LIN {X 0,Y 397.096,Z 510.019,A -85,B 0,C 180,E1 -11203.649,E2 -11203.649} C_VEL
LIN {X 0,Y 397.1,Z 510.023,A -85,B 0,C 180,E1 -11206.521,E2 -11206.521} C_VEL
LIN {X 0,Y 397.111,Z 510.021,A -85,B 0,C 180,E1 -11210.424,E2 -11210.424} C_VEL
LIN {X 0,Y 397.107,Z 510.02,A -85,B 0,C 180,E1 -11214.266,E2 -11214.266} C_VEL
LIN {X 0,Y 397.113,Z 510.025,A -85,B 0,C 180,E1 -11216.728,E2 -11216.728} C_VEL
LIN {X 0,Y 397.129,Z 510.185,A -85,B 0,C 180,E1 -11218.395,E2 -11218.395} C_VEL
LIN {X 0,Y 399.849,Z 521.047,A -85,B 0,C 180,E1 -11221.067,E2 -11221.067} C_VEL
LIN {X 0,Y 401.622,Z 530.428,A -85,B 0,C 180,E1 -11223.183,E2 -11223.183} C_VEL
LIN {X 0,Y 401.493,Z 534.696,A -85,B 0,C 180,E1 -11224.049,E2 -11224.049} C_VEL
LIN {X 0,Y 399.863,Z 552.668,A -85,B 0,C 180,E1 -11227.526,E2 -11227.526} C_VEL
LIN {X 0,Y 399.207,Z 561.982,A -85,B 0,C 180,E1 -11229.268,E2 -11229.268} C_VEL
LIN {X 0,Y 402.568,Z 583.232,A -85,B 0,C 180,E1 -11230.004,E2 -11230.004} C_VEL
LIN {X 0,Y 404.122,Z 598.929,A -85,B 0,C 180,E1 -11230.474,E2 -11230.474} C_VEL
LIN {X 0,Y 402.335,Z 674.306,A -85,B 0,C 180,E1 -11232.135,E2 -11232.135} C_VEL
LIN {X 0,Y 401.685,Z 687.799,A -85,B 0,C 180,E1 -11232.631,E2 -11232.631} C_VEL
LIN {X 0,Y 400.492,Z 707.778,A -85,B 0,C 180,E1 -11233.694,E2 -11233.694} C_VEL
LIN {X 0,Y 399.642,Z 720.158,A -85,B 0,C 180,E1 -11234.575,E2 -11234.575} C_VEL
LIN {X 0,Y 398.904,Z 731.177,A -85,B 0,C 180,E1 -11235.59,E2 -11235.59} C_VEL
LIN {X 0,Y 398.092,Z 741.058,A -85,B 0,C 180,E1 -11236.732,E2 -11236.732} C_VEL
LIN {X 0,Y 397.429,Z 750.03,A -85,B 0,C 180,E1 -11238.008,E2 -11238.008} C_VEL
LIN {X 0,Y 396.786,Z 758.764,A -85,B 0,C 180,E1 -11239.54,E2 -11239.54} C_VEL
LIN {X 0,Y 396.358,Z 765.698,A -85,B 0,C 180,E1 -11241.075,E2 -11241.075} C_VEL
LIN {X 0,Y 396.008,Z 772.039,A -85,B 0,C 180,E1 -11242.864,E2 -11242.864} C_VEL
LIN {X 0,Y 395.867,Z 776.173,A -85,B 0,C 180,E1 -11244.397,E2 -11244.397} C_VEL
LIN {X 0,Y 395.803,Z 779.229,A -85,B 0,C 180,E1 -11245.927,E2 -11245.927} C_VEL
LIN {X 0,Y 395.793,Z 780.728,A -85,B 0,C 180,E1 -11246.946,E2 -11246.946} C_VEL
LIN {X 0,Y 395.838,Z 781.772,A -85,B 0,C 180,E1 -11247.965,E2 -11247.965} C_VEL
LIN {X 0,Y 395.803,Z 782.42,A -85,B 0,C 180,E1 -11248.983,E2 -11248.983} C_VEL
LIN {X 0,Y 395.787,Z 782.679,A -85,B 0,C 180,E1 -11250,E2 -11250} C_VEL
LIN {X 0,Y 395.803,Z 782.515,A -85,B 0,C 180,E1 -11251.017,E2 -11251.017} C_VEL
LIN {X 0,Y 395.838,Z 781.93,A -85,B 0,C 180,E1 -11252.035,E2 -11252.035} C_VEL
LIN {X 0,Y 395.805,Z 779.574,A -85,B 0,C 180,E1 -11254.073,E2 -11254.073} C_VEL
LIN {X 0,Y 395.871,Z 776.658,A -85,B 0,C 180,E1 -11255.603,E2 -11255.603} C_VEL
LIN {X 0,Y 396.025,Z 772.695,A -85,B 0,C 180,E1 -11257.136,E2 -11257.136} C_VEL
LIN {X 0,Y 396.366,Z 766.556,A -85,B 0,C 180,E1 -11258.925,E2 -11258.925} C_VEL
LIN {X 0,Y 396.849,Z 759.844,A -85,B 0,C 180,E1 -11260.458,E2 -11260.458} C_VEL
LIN {X 0,Y 397.523,Z 751.498,A -85,B 0,C 180,E1 -11261.989,E2 -11261.989} C_VEL
LIN {X 0,Y 398.233,Z 742.869,A -85,B 0,C 180,E1 -11263.263,E2 -11263.263} C_VEL
LIN {X 0,Y 399.082,Z 732.464,A -85,B 0,C 180,E1 -11264.507,E2 -11264.507} C_VEL
LIN {X 0,Y 399.924,Z 721.614,A -85,B 0,C 180,E1 -11265.545,E2 -11265.545} C_VEL
LIN {X 0,Y 400.746,Z 709.682,A -85,B 0,C 180,E1 -11266.426,E2 -11266.426} C_VEL
LIN {X 0,Y 401.51,Z 697.234,A -85,B 0,C 180,E1 -11267.114,E2 -11267.114} C_VEL
LIN {X 0,Y 402.075,Z 685.131,A -85,B 0,C 180,E1 -11267.581,E2 -11267.581} C_VEL
LIN {X 0,Y 402.418,Z 671.595,A -85,B 0,C 180,E1 -11267.894,E2 -11267.894} C_VEL
LIN {X 0,Y 403.196,Z 596.853,A -85,B 0,C 180,E1 -11269.234,E2 -11269.234} C_VEL
LIN {X 0,Y 398.792,Z 564.219,A -85,B 0,C 180,E1 -11270.099,E2 -11270.099} C_VEL
LIN {X 0,Y 400.137,Z 545.377,A -85,B 0,C 180,E1 -11273.551,E2 -11273.551} C_VEL
LIN {X 0,Y 401.205,Z 530.505,A -85,B 0,C 180,E1 -11276.307,E2 -11276.307} C_VEL
LIN {X 0,Y 399.773,Z 522.21,A -85,B 0,C 180,E1 -11277.971,E2 -11277.971} C_VEL
LIN {X 0,Y 397.11,Z 510.021,A -85,B 0,C 180,E1 -11280.533,E2 -11280.533} C_VEL
LIN {X 0,Y 397.123,Z 510.017,A -85,B 0,C 180,E1 -11284.493,E2 -11284.493} C_VEL
LIN {X 0,Y 397.101,Z 509.992,A -85,B 0,C 180,E1 -11288.274,E2 -11288.274} C_VEL
LIN {X 0,Y 397.087,Z 510.02,A -85,B 0,C 180,E1 -11290.908,E2 -11290.908} C_VEL
LIN {X 0,Y 397.1,Z 510.015,A -85,B 0,C 180,E1 -11293.647,E2 -11293.647} C_VEL
LIN {X 0,Y 397.099,Z 510.02,A -85,B 0,C 180,E1 -11296.52,E2 -11296.52} C_VEL
LIN {X 0,Y 397.115,Z 510.019,A -85,B 0,C 180,E1 -11299.551,E2 -11299.551} C_VEL
LIN {X 0,Y 397.093,Z 510.016,A -85,B 0,C 180,E1 -11302.789,E2 -11302.789} C_VEL
LIN {X 0,Y 397.112,Z 510.016,A -85,B 0,C 180,E1 -11306.282,E2 -11306.282} C_VEL
LIN {X 0,Y 397.107,Z 510.009,A -85,B 0,C 180,E1 -11310.133,E2 -11310.133} C_VEL
LIN {X 0,Y 397.188,Z 510.008,A -85,B 0,C 180,E1 -11312.609,E2 -11312.609} C_VEL
LIN {X 0,Y 397.121,Z 509.998,A -85,B 0,C 180,E1 -11315.981,E2 -11315.981} C_VEL
LIN {X 0,Y 397.13,Z 510.014,A -85,B 0,C 180,E1 -11319.704,E2 -11319.704} C_VEL
LIN {X 0,Y 397.173,Z 509.997,A -85,B 0,C 180,E1 -11322.845,E2 -11322.845} C_VEL
LIN {X 0,Y 397.22,Z 510.003,A -85,B 0,C 180,E1 -11326.703,E2 -11326.703} C_VEL
LIN {X 0,Y 397.221,Z 509.995,A -85,B 0,C 180,E1 -11329.809,E2 -11329.809} C_VEL
LIN {X 0,Y 397.349,Z 509.974,A -85,B 0,C 180,E1 -11332.888,E2 -11332.888} C_VEL
LIN {X 0,Y 397.254,Z 510,A -85,B 0,C 180,E1 -11334.925,E2 -11334.925} C_VEL
LIN {X 0,Y 397.443,Z 509.969,A -85,B 0,C 180,E1 -11337.973,E2 -11337.973} C_VEL
LIN {X 0,Y 397.574,Z 509.937,A -85,B 0,C 180,E1 -11340,E2 -11340} C_VEL
LIN {X 0,Y 397.376,Z 509.984,A -85,B 0,C 180,E1 -11343.042,E2 -11343.042} C_VEL
LIN {X 0,Y 397.345,Z 509.978,A -85,B 0,C 180,E1 -11346.602,E2 -11346.602} C_VEL
LIN {X 0,Y 397.245,Z 509.987,A -85,B 0,C 180,E1 -11349.162,E2 -11349.162} C_VEL
LIN {X 0,Y 397.212,Z 510.004,A -85,B 0,C 180,E1 -11352.259,E2 -11352.259} C_VEL
LIN {X 0,Y 397.171,Z 509.995,A -85,B 0,C 180,E1 -11355.393,E2 -11355.393} C_VEL
LIN {X 0,Y 397.155,Z 510.008,A -85,B 0,C 180,E1 -11358.574,E2 -11358.574} C_VEL
LIN {X 0,Y 397.09,Z 510.013,A -85,B 0,C 180,E1 -11361.819,E2 -11361.819} C_VEL
LIN {X 0,Y 397.15,Z 510.011,A -85,B 0,C 180,E1 -11365.132,E2 -11365.132} C_VEL
LIN {X 0,Y 397.158,Z 510.008,A -85,B 0,C 180,E1 -11367.777,E2 -11367.777} C_VEL
LIN {X 0,Y 397.083,Z 510.017,A -85,B 0,C 180,E1 -11370.883,E2 -11370.883} C_VEL
LIN {X 0,Y 397.121,Z 510.013,A -85,B 0,C 180,E1 -11374.494,E2 -11374.494} C_VEL
LIN {X 0,Y 397.102,Z 510.02,A -85,B 0,C 180,E1 -11378.276,E2 -11378.276} C_VEL
LIN {X 0,Y 397.086,Z 510.024,A -85,B 0,C 180,E1 -11380.91,E2 -11380.91} C_VEL
LIN {X 0,Y 397.102,Z 510.017,A -85,B 0,C 180,E1 -11383.649,E2 -11383.649} C_VEL
LIN {X 0,Y 397.104,Z 510.02,A -85,B 0,C 180,E1 -11386.521,E2 -11386.521} C_VEL
LIN {X 0,Y 397.113,Z 510.017,A -85,B 0,C 180,E1 -11390.424,E2 -11390.424} C_VEL
LIN {X 0,Y 397.108,Z 510.016,A -85,B 0,C 180,E1 -11394.266,E2 -11394.266} C_VEL
LIN {X 0,Y 397.115,Z 510.021,A -85,B 0,C 180,E1 -11396.728,E2 -11396.728} C_VEL
LIN {X 0,Y 397.153,Z 510.107,A -85,B 0,C 180,E1 -11400.481,E2 -11400.481} C_VEL
LIN {X 0,Y 399.874,Z 522.345,A -85,B 0,C 180,E1 -11403.03,E2 -11403.03} C_VEL
LIN {X 0,Y 400.773,Z 528.562,A -85,B 0,C 180,E1 -11404.278,E2 -11404.278} C_VEL
LIN {X 0,Y 399.987,Z 546.3,A -85,B 0,C 180,E1 -11407.506,E2 -11407.506} C_VEL
LIN {X 0,Y 399.916,Z 548.272,A -85,B 0,C 180,E1 -11407.847,E2 -11407.847} C_VEL
LIN {X 0,Y 404.133,Z 570.893,A -85,B 0,C 180,E1 -11408.514,E2 -11408.514} C_VEL
LIN {X 0,Y 402.844,Z 658.693,A -85,B 0,C 180,E1 -11410.112,E2 -11410.112} C_VEL
LIN {X 0,Y 402.388,Z 671.82,A -85,B 0,C 180,E1 -11410.553,E2 -11410.553} C_VEL
LIN {X 0,Y 401.815,Z 684.753,A -85,B 0,C 180,E1 -11411.216,E2 -11411.216} C_VEL
LIN {X 0,Y 401.115,Z 696.348,A -85,B 0,C 180,E1 -11412.013,E2 -11412.013} C_VEL
LIN {X 0,Y 400.193,Z 707.742,A -85,B 0,C 180,E1 -11413.025,E2 -11413.025} C_VEL
LIN {X 0,Y 399.274,Z 717.987,A -85,B 0,C 180,E1 -11414.168,E2 -11414.168} C_VEL
LIN {X 0,Y 398.43,Z 727.248,A -85,B 0,C 180,E1 -11415.442,E2 -11415.442} C_VEL
LIN {X 0,Y 397.704,Z 736.147,A -85,B 0,C 180,E1 -11416.979,E2 -11416.979} C_VEL
LIN {X 0,Y 397.034,Z 743.308,A -85,B 0,C 180,E1 -11418.514,E2 -11418.514} C_VEL
LIN {X 0,Y 396.477,Z 749.856,A -85,B 0,C 180,E1 -11420.306,E2 -11420.306} C_VEL
LIN {X 0,Y 396.179,Z 754.149,A -85,B 0,C 180,E1 -11421.841,E2 -11421.841} C_VEL
LIN {X 0,Y 395.935,Z 757.992,A -85,B 0,C 180,E1 -11423.737,E2 -11423.737} C_VEL
LIN {X 0,Y 395.861,Z 759.623,A -85,B 0,C 180,E1 -11424.907,E2 -11424.907} C_VEL
LIN {X 0,Y 395.752,Z 761.187,A -85,B 0,C 180,E1 -11426.946,E2 -11426.946} C_VEL
LIN {X 0,Y 395.81,Z 761.386,A -85,B 0,C 180,E1 -11427.965,E2 -11427.965} C_VEL
LIN {X 0,Y 395.797,Z 761.157,A -85,B 0,C 180,E1 -11428.983,E2 -11428.983} C_VEL
LIN {X 0,Y 395.808,Z 759.558,A -85,B 0,C 180,E1 -11431.017,E2 -11431.017} C_VEL
LIN {X 0,Y 395.864,Z 758.807,A -85,B 0,C 180,E1 -11431.558,E2 -11431.558} C_VEL
LIN {X 0,Y 395.29,Z 757.58,A -85,B 0,C 180,E1 -11432.391,E2 -11432.391} C_VEL
LIN {X 0,Y 392.536,Z 755.077,A -85,B 0,C 180,E1 -11433.732,E2 -11433.732} C_VEL
LIN {X 0,Y 389.848,Z 751.866,A -85,B 0,C 180,E1 -11435.055,E2 -11435.055} C_VEL
LIN {X 0,Y 389.388,Z 749.468,A -85,B 0,C 180,E1 -11435.85,E2 -11435.85} C_VEL
LIN {X 0,Y 389.891,Z 743.419,A -85,B 0,C 180,E1 -11437.513,E2 -11437.513} C_VEL
LIN {X 0,Y 390.438,Z 736.304,A -85,B 0,C 180,E1 -11439.062,E2 -11439.062} C_VEL
LIN {X 0,Y 391.27,Z 727.439,A -85,B 0,C 180,E1 -11440.609,E2 -11440.609} C_VEL
LIN {X 0,Y 392.214,Z 717.208,A -85,B 0,C 180,E1 -11442.023,E2 -11442.023} C_VEL
LIN {X 0,Y 392.981,Z 706.853,A -85,B 0,C 180,E1 -11443.18,E2 -11443.18} C_VEL
LIN {X 0,Y 393.927,Z 695.167,A -85,B 0,C 180,E1 -11444.2,E2 -11444.2} C_VEL
LIN {X 0,Y 394.595,Z 683.906,A -85,B 0,C 180,E1 -11444.966,E2 -11444.966} C_VEL
LIN {X 0,Y 395.122,Z 671.335,A -85,B 0,C 180,E1 -11445.607,E2 -11445.607} C_VEL
LIN {X 0,Y 395.536,Z 658.217,A -85,B 0,C 180,E1 -11446.044,E2 -11446.044} C_VEL
LIN {X 0,Y 396.696,Z 571.194,A -85,B 0,C 180,E1 -11447.648,E2 -11447.648} C_VEL
LIN {X 0,Y 392.7,Z 548.444,A -85,B 0,C 180,E1 -11448.291,E2 -11448.291} C_VEL
LIN {X 0,Y 393.475,Z 530.342,A -85,B 0,C 180,E1 -11451.579,E2 -11451.579} C_VEL
LIN {X 0,Y 393.57,Z 527.947,A -85,B 0,C 180,E1 -11452.024,E2 -11452.024} C_VEL
LIN {X 0,Y 390.969,Z 514.765,A -85,B 0,C 180,E1 -11454.704,E2 -11454.704} C_VEL
LIN {X 0,Y 390.13,Z 510.894,A -85,B 0,C 180,E1 -11455.544,E2 -11455.544} C_VEL
LIN {X 0,Y 390.099,Z 510.893,A -85,B 0,C 180,E1 -11458.019,E2 -11458.019} C_VEL
LIN {X 0,Y 390.025,Z 510.904,A -85,B 0,C 180,E1 -11461.503,E2 -11461.503} C_VEL
LIN {X 0,Y 390.085,Z 510.895,A -85,B 0,C 180,E1 -11465.206,E2 -11465.206} C_VEL
LIN {X 0,Y 390.068,Z 510.893,A -85,B 0,C 180,E1 -11469.217,E2 -11469.217} C_VEL
LIN {X 0,Y 390.114,Z 510.89,A -85,B 0,C 180,E1 -11472.385,E2 -11472.385} C_VEL
LIN {X 0,Y 390.061,Z 510.887,A -85,B 0,C 180,E1 -11475.356,E2 -11475.356} C_VEL
LIN {X 0,Y 390.03,Z 510.9,A -85,B 0,C 180,E1 -11478.186,E2 -11478.186} C_VEL
LIN {X 0,Y 390.088,Z 510.897,A -85,B 0,C 180,E1 -11480.907,E2 -11480.907} C_VEL
LIN {X 0,Y 390.052,Z 510.899,A -85,B 0,C 180,E1 -11484.044,E2 -11484.044} C_VEL
LIN {X 0,Y 396.302,Z 528.476,A -85,B 0,C 180,E1 -11484.733,E2 -11484.733} C_VEL
LIN {X 0,Y 394.645,Z 615.636,A -85,B 0,C 180,E1 -11486.587,E2 -11486.587} C_VEL
LIN {X 0,Y 394.295,Z 629.503,A -85,B 0,C 180,E1 -11487.103,E2 -11487.103} C_VEL
LIN {X 0,Y 393.79,Z 641.997,A -85,B 0,C 180,E1 -11487.779,E2 -11487.779} C_VEL
LIN {X 0,Y 393.143,Z 653.763,A -85,B 0,C 180,E1 -11488.624,E2 -11488.624} C_VEL
LIN {X 0,Y 392.462,Z 665.327,A -85,B 0,C 180,E1 -11489.68,E2 -11489.68} C_VEL
LIN {X 0,Y 391.78,Z 675.774,A -85,B 0,C 180,E1 -11490.883,E2 -11490.883} C_VEL
LIN {X 0,Y 391.124,Z 684.741,A -85,B 0,C 180,E1 -11492.148,E2 -11492.148} C_VEL
LIN {X 0,Y 390.524,Z 692.947,A -85,B 0,C 180,E1 -11493.558,E2 -11493.558} C_VEL
LIN {X 0,Y 390.07,Z 699.565,A -85,B 0,C 180,E1 -11494.95,E2 -11494.95} C_VEL
LIN {X 0,Y 389.656,Z 705.939,A -85,B 0,C 180,E1 -11496.621,E2 -11496.621} C_VEL
LIN {X 0,Y 389.324,Z 710.824,A -85,B 0,C 180,E1 -11498.28,E2 -11498.28} C_VEL
LIN {X 0,Y 389.08,Z 714.432,A -85,B 0,C 180,E1 -11499.928,E2 -11499.928} C_VEL
LIN {X 0,Y 388.956,Z 716.211,A -85,B 0,C 180,E1 -11501.02,E2 -11501.02} C_VEL
LIN {X 0,Y 388.919,Z 717.475,A -85,B 0,C 180,E1 -11502.109,E2 -11502.109} C_VEL
LIN {X 0,Y 388.914,Z 718.323,A -85,B 0,C 180,E1 -11503.282,E2 -11503.282} C_VEL
LIN {X 0,Y 388.894,Z 718.649,A -85,B 0,C 180,E1 -11504.271,E2 -11504.271} C_VEL
LIN {X 0,Y 388.915,Z 718.545,A -85,B 0,C 180,E1 -11505.345,E2 -11505.345} C_VEL
LIN {X 0,Y 389.103,Z 717.267,A -85,B 0,C 180,E1 -11507.246,E2 -11507.246} C_VEL
LIN {X 0,Y 389.283,Z 715.597,A -85,B 0,C 180,E1 -11508.545,E2 -11508.545} C_VEL
LIN {X 0,Y 389.597,Z 712.589,A -85,B 0,C 180,E1 -11510.132,E2 -11510.132} C_VEL
LIN {X 0,Y 390.022,Z 708.477,A -85,B 0,C 180,E1 -11511.711,E2 -11511.711} C_VEL
LIN {X 0,Y 390.644,Z 702.159,A -85,B 0,C 180,E1 -11513.544,E2 -11513.544} C_VEL
LIN {X 0,Y 391.31,Z 695.239,A -85,B 0,C 180,E1 -11515.106,E2 -11515.106} C_VEL
LIN {X 0,Y 392.074,Z 686.569,A -85,B 0,C 180,E1 -11516.66,E2 -11516.66} C_VEL
LIN {X 0,Y 393.011,Z 677.655,A -85,B 0,C 180,E1 -11517.95,E2 -11517.95} C_VEL
LIN {X 0,Y 393.661,Z 669.12,A -85,B 0,C 180,E1 -11518.977,E2 -11518.977} C_VEL
LIN {X 0,Y 394.55,Z 658.678,A -85,B 0,C 180,E1 -11520,E2 -11520} C_VEL
LIN {X 0,Y 395.336,Z 647.141,A -85,B 0,C 180,E1 -11520.891,E2 -11520.891} C_VEL
LIN {X 0,Y 395.963,Z 634.266,A -85,B 0,C 180,E1 -11521.653,E2 -11521.653} C_VEL
LIN {X 0,Y 396.404,Z 621.296,A -85,B 0,C 180,E1 -11522.191,E2 -11522.191} C_VEL
LIN {X 0,Y 396.817,Z 602.346,A -85,B 0,C 180,E1 -11522.664,E2 -11522.664} C_VEL
LIN {X 0,Y 398.824,Z 531.552,A -85,B 0,C 180,E1 -11524.273,E2 -11524.273} C_VEL
LIN {X 0,Y 393.097,Z 518.551,A -85,B 0,C 180,E1 -11525.032,E2 -11525.032} C_VEL
LIN {X 0,Y 390.773,Z 513.32,A -85,B 0,C 180,E1 -11525.353,E2 -11525.353} C_VEL
LIN {X 0,Y 390.332,Z 510.866,A -85,B 0,C 180,E1 -11526.202,E2 -11526.202} C_VEL
LIN {X 0,Y 390.307,Z 510.868,A -85,B 0,C 180,E1 -11528.282,E2 -11528.282} C_VEL
LIN {X 0,Y 390.171,Z 510.883,A -85,B 0,C 180,E1 -11532.483,E2 -11532.483} C_VEL
LIN {X 0,Y 390.132,Z 510.89,A -85,B 0,C 180,E1 -11535.677,E2 -11535.677} C_VEL
LIN {X 0,Y 390.097,Z 510.894,A -85,B 0,C 180,E1 -11538.922,E2 -11538.922} C_VEL
LIN {X 0,Y 390.032,Z 510.899,A -85,B 0,C 180,E1 -11542.234,E2 -11542.234} C_VEL
LIN {X 0,Y 390.112,Z 510.887,A -85,B 0,C 180,E1 -11545.744,E2 -11545.744} C_VEL
LIN {X 0,Y 390.059,Z 510.895,A -85,B 0,C 180,E1 -11549.109,E2 -11549.109} C_VEL
LIN {X 0,Y 390.037,Z 510.897,A -85,B 0,C 180,E1 -11552.722,E2 -11552.722} C_VEL
LIN {X 0,Y 390.051,Z 510.893,A -85,B 0,C 180,E1 -11555.826,E2 -11555.826} C_VEL
LIN {X 0,Y 390.066,Z 510.898,A -85,B 0,C 180,E1 -11559.219,E2 -11559.219} C_VEL
LIN {X 0,Y 390.037,Z 510.898,A -85,B 0,C 180,E1 -11562.375,E2 -11562.375} C_VEL
LIN {X 0,Y 390.042,Z 510.9,A -85,B 0,C 180,E1 -11565.355,E2 -11565.355} C_VEL
LIN {X 0,Y 390.029,Z 510.903,A -85,B 0,C 180,E1 -11568.188,E2 -11568.188} C_VEL
LIN {X 0,Y 390.089,Z 510.897,A -85,B 0,C 180,E1 -11570.909,E2 -11570.909} C_VEL
LIN {X 0,Y 390.083,Z 510.898,A -85,B 0,C 180,E1 -11574.794,E2 -11574.794} C_VEL
LIN {X 0,Y 390.067,Z 511.059,A -85,B 0,C 180,E1 -11577.867,E2 -11577.867} C_VEL
LIN {X 0,Y 392.715,Z 521.386,A -85,B 0,C 180,E1 -11580.52,E2 -11580.52} C_VEL
LIN {X 0,Y 394.721,Z 531.57,A -85,B 0,C 180,E1 -11582.905,E2 -11582.905} C_VEL
LIN {X 0,Y 394.82,Z 534.729,A -85,B 0,C 180,E1 -11583.577,E2 -11583.577} C_VEL
LIN {X 0,Y 393.103,Z 552.575,A -85,B 0,C 180,E1 -11587.117,E2 -11587.117} C_VEL
LIN {X 0,Y 392.389,Z 560.982,A -85,B 0,C 180,E1 -11588.745,E2 -11588.745} C_VEL
LIN {X 0,Y 395.402,Z 579.122,A -85,B 0,C 180,E1 -11589.437,E2 -11589.437} C_VEL
LIN {X 0,Y 397.597,Z 598.765,A -85,B 0,C 180,E1 -11590.07,E2 -11590.07} C_VEL
LIN {X 0,Y 395.708,Z 673.591,A -85,B 0,C 180,E1 -11591.759,E2 -11591.759} C_VEL
LIN {X 0,Y 395.043,Z 686.973,A -85,B 0,C 180,E1 -11592.263,E2 -11592.263} C_VEL
LIN {X 0,Y 394.15,Z 698.816,A -85,B 0,C 180,E1 -11592.89,E2 -11592.89} C_VEL
LIN {X 0,Y 393.233,Z 713.143,A -85,B 0,C 180,E1 -11593.785,E2 -11593.785} C_VEL
LIN {X 0,Y 392.421,Z 724.245,A -85,B 0,C 180,E1 -11594.683,E2 -11594.683} C_VEL
LIN {X 0,Y 391.686,Z 734.793,A -85,B 0,C 180,E1 -11595.763,E2 -11595.763} C_VEL
LIN {X 0,Y 390.902,Z 744.598,A -85,B 0,C 180,E1 -11597.013,E2 -11597.013} C_VEL
LIN {X 0,Y 390.056,Z 754.376,A -85,B 0,C 180,E1 -11598.569,E2 -11598.569} C_VEL
LIN {X 0,Y 389.477,Z 762.174,A -85,B 0,C 180,E1 -11600.13,E2 -11600.13} C_VEL
LIN {X 0,Y 389.126,Z 768.388,A -85,B 0,C 180,E1 -11601.693,E2 -11601.693} C_VEL
LIN {X 0,Y 388.903,Z 773.307,A -85,B 0,C 180,E1 -11603.254,E2 -11603.254} C_VEL
LIN {X 0,Y 388.786,Z 777.078,A -85,B 0,C 180,E1 -11604.814,E2 -11604.814} C_VEL
LIN {X 0,Y 388.728,Z 779.015,A -85,B 0,C 180,E1 -11605.853,E2 -11605.853} C_VEL
LIN {X 0,Y 388.696,Z 780.522,A -85,B 0,C 180,E1 -11606.891,E2 -11606.891} C_VEL
LIN {X 0,Y 388.736,Z 781.571,A -85,B 0,C 180,E1 -11607.928,E2 -11607.928} C_VEL
LIN {X 0,Y 388.734,Z 782.224,A -85,B 0,C 180,E1 -11608.964,E2 -11608.964} C_VEL
LIN {X 0,Y 388.716,Z 782.486,A -85,B 0,C 180,E1 -11610,E2 -11610} C_VEL
LIN {X 0,Y 388.716,Z 782.331,A -85,B 0,C 180,E1 -11611.036,E2 -11611.036} C_VEL
LIN {X 0,Y 388.736,Z 781.75,A -85,B 0,C 180,E1 -11612.072,E2 -11612.072} C_VEL
LIN {X 0,Y 388.729,Z 779.403,A -85,B 0,C 180,E1 -11614.147,E2 -11614.147} C_VEL
LIN {X 0,Y 388.786,Z 776.201,A -85,B 0,C 180,E1 -11615.84,E2 -11615.84} C_VEL
LIN {X 0,Y 389.057,Z 770.95,A -85,B 0,C 180,E1 -11617.786,E2 -11617.786} C_VEL
LIN {X 0,Y 389.375,Z 765.411,A -85,B 0,C 180,E1 -11619.349,E2 -11619.349} C_VEL
LIN {X 0,Y 389.87,Z 758.481,A -85,B 0,C 180,E1 -11620.91,E2 -11620.91} C_VEL
LIN {X 0,Y 390.69,Z 749.779,A -85,B 0,C 180,E1 -11622.466,E2 -11622.466} C_VEL
LIN {X 0,Y 391.538,Z 739.805,A -85,B 0,C 180,E1 -11623.9,E2 -11623.9} C_VEL
LIN {X 0,Y 392.364,Z 729.739,A -85,B 0,C 180,E1 -11625.053,E2 -11625.053} C_VEL
LIN {X 0,Y 393.31,Z 718.48,A -85,B 0,C 180,E1 -11626.079,E2 -11626.079} C_VEL
LIN {X 0,Y 394.148,Z 706.772,A -85,B 0,C 180,E1 -11626.909,E2 -11626.909} C_VEL
LIN {X 0,Y 394.892,Z 693.826,A -85,B 0,C 180,E1 -11627.577,E2 -11627.577} C_VEL
LIN {X 0,Y 395.426,Z 681.051,A -85,B 0,C 180,E1 -11628.021,E2 -11628.021} C_VEL
LIN {X 0,Y 396.055,Z 642.822,A -85,B 0,C 180,E1 -11628.743,E2 -11628.743} C_VEL
LIN {X 0,Y 396.517,Z 597.684,A -85,B 0,C 180,E1 -11629.569,E2 -11629.569} C_VEL
LIN {X 0,Y 391.887,Z 563.247,A -85,B 0,C 180,E1 -11630.503,E2 -11630.503} C_VEL
LIN {X 0,Y 393.402,Z 542.69,A -85,B 0,C 180,E1 -11634.342,E2 -11634.342} C_VEL
LIN {X 0,Y 394.226,Z 531.472,A -85,B 0,C 180,E1 -11636.466,E2 -11636.466} C_VEL
LIN {X 0,Y 392.676,Z 522.867,A -85,B 0,C 180,E1 -11638.231,E2 -11638.231} C_VEL
LIN {X 0,Y 390.076,Z 510.898,A -85,B 0,C 180,E1 -11640.782,E2 -11640.782} C_VEL
LIN {X 0,Y 390.066,Z 510.896,A -85,B 0,C 180,E1 -11644.024,E2 -11644.024} C_VEL
LIN {X 0,Y 390.041,Z 510.873,A -85,B 0,C 180,E1 -11647.55,E2 -11647.55} C_VEL
LIN {X 0,Y 390.054,Z 510.895,A -85,B 0,C 180,E1 -11650.821,E2 -11650.821} C_VEL
LIN {X 0,Y 390.053,Z 510.892,A -85,B 0,C 180,E1 -11653.886,E2 -11653.886} C_VEL
LIN {X 0,Y 390.075,Z 510.887,A -85,B 0,C 180,E1 -11657.619,E2 -11657.619} C_VEL
LIN {X 0,Y 390.089,Z 510.895,A -85,B 0,C 180,E1 -11660.908,E2 -11660.908} C_VEL
LIN {X 0,Y 390.079,Z 510.889,A -85,B 0,C 180,E1 -11664.793,E2 -11664.793} C_VEL
LIN {X 0,Y 390.021,Z 510.895,A -85,B 0,C 180,E1 -11668.495,E2 -11668.495} C_VEL
LIN {X 0,Y 390.11,Z 510.888,A -85,B 0,C 180,E1 -11672.07,E2 -11672.07} C_VEL
LIN {X 0,Y 390.069,Z 510.878,A -85,B 0,C 180,E1 -11675.519,E2 -11675.519} C_VEL
LIN {X 0,Y 390.079,Z 510.894,A -85,B 0,C 180,E1 -11679.53,E2 -11679.53} C_VEL
LIN {X 0,Y 390.129,Z 510.871,A -85,B 0,C 180,E1 -11683.248,E2 -11683.248} C_VEL
LIN {X 0,Y 390.186,Z 510.878,A -85,B 0,C 180,E1 -11686.561,E2 -11686.561} C_VEL
LIN {X 0,Y 390.17,Z 510.874,A -85,B 0,C 180,E1 -11689.623,E2 -11689.623} C_VEL
LIN {X 0,Y 390.299,Z 510.85,A -85,B 0,C 180,E1 -11692.759,E2 -11692.759} C_VEL
LIN {X 0,Y 390.226,Z 510.874,A -85,B 0,C 180,E1 -11694.834,E2 -11694.834} C_VEL
LIN {X 0,Y 390.412,Z 510.845,A -85,B 0,C 180,E1 -11697.937,E2 -11697.937} C_VEL
LIN {X 0,Y 390.543,Z 510.812,A -85,B 0,C 180,E1 -11700,E2 -11700} C_VEL
LIN {X 0,Y 390.31,Z 510.865,A -85,B 0,C 180,E1 -11703.097,E2 -11703.097} C_VEL
LIN {X 0,Y 390.301,Z 510.855,A -85,B 0,C 180,E1 -11706.595,E2 -11706.595} C_VEL
LIN {X 0,Y 390.197,Z 510.866,A -85,B 0,C 180,E1 -11709.329,E2 -11709.329} C_VEL
LIN {X 0,Y 390.163,Z 510.883,A -85,B 0,C 180,E1 -11712.484,E2 -11712.484} C_VEL
LIN {X 0,Y 390.131,Z 510.869,A -85,B 0,C 180,E1 -11715.678,E2 -11715.678} C_VEL
LIN {X 0,Y 390.098,Z 510.891,A -85,B 0,C 180,E1 -11718.923,E2 -11718.923} C_VEL
LIN {X 0,Y 390.033,Z 510.892,A -85,B 0,C 180,E1 -11722.235,E2 -11722.235} C_VEL
LIN {X 0,Y 390.113,Z 510.889,A -85,B 0,C 180,E1 -11725.744,E2 -11725.744} C_VEL
LIN {X 0,Y 390.06,Z 510.887,A -85,B 0,C 180,E1 -11729.11,E2 -11729.11} C_VEL
LIN {X 0,Y 390.051,Z 510.9,A -85,B 0,C 180,E1 -11732.721,E2 -11732.721} C_VEL
LIN {X 0,Y 390.053,Z 510.895,A -85,B 0,C 180,E1 -11735.827,E2 -11735.827} C_VEL
LIN {X 0,Y 390.068,Z 510.893,A -85,B 0,C 180,E1 -11739.22,E2 -11739.22} C_VEL
LIN {X 0,Y 390.041,Z 510.902,A -85,B 0,C 180,E1 -11742.375,E2 -11742.375} C_VEL
LIN {X 0,Y 390.047,Z 510.901,A -85,B 0,C 180,E1 -11745.356,E2 -11745.356} C_VEL
LIN {X 0,Y 390.031,Z 510.9,A -85,B 0,C 180,E1 -11748.188,E2 -11748.188} C_VEL
LIN {X 0,Y 390.09,Z 510.897,A -85,B 0,C 180,E1 -11750.909,E2 -11750.909} C_VEL
LIN {X 0,Y 390.085,Z 510.887,A -85,B 0,C 180,E1 -11754.794,E2 -11754.794} C_VEL
LIN {X 0,Y 390.024,Z 510.897,A -85,B 0,C 180,E1 -11758.497,E2 -11758.497} C_VEL
LIN {X 0,Y 390.083,Z 510.96,A -85,B 0,C 180,E1 -11760.141,E2 -11760.141} C_VEL
LIN {X 0,Y 392.702,Z 522.391,A -85,B 0,C 180,E1 -11762.56,E2 -11762.56} C_VEL
LIN {X 0,Y 393.918,Z 529.866,A -85,B 0,C 180,E1 -11764.081,E2 -11764.081} C_VEL
LIN {X 0,Y 393.122,Z 547.663,A -85,B 0,C 180,E1 -11767.341,E2 -11767.341} C_VEL
LIN {X 0,Y 393.123,Z 548.442,A -85,B 0,C 180,E1 -11767.478,E2 -11767.478} C_VEL
LIN {X 0,Y 397.43,Z 571.422,A -85,B 0,C 180,E1 -11768.165,E2 -11768.165} C_VEL
LIN {X 0,Y 396.152,Z 657.933,A -85,B 0,C 180,E1 -11769.761,E2 -11769.761} C_VEL
LIN {X 0,Y 395.713,Z 670.691,A -85,B 0,C 180,E1 -11770.178,E2 -11770.178} C_VEL
LIN {X 0,Y 395.153,Z 683.49,A -85,B 0,C 180,E1 -11770.82,E2 -11770.82} C_VEL
LIN {X 0,Y 394.427,Z 694.544,A -85,B 0,C 180,E1 -11771.563,E2 -11771.563} C_VEL
LIN {X 0,Y 393.501,Z 706.451,A -85,B 0,C 180,E1 -11772.593,E2 -11772.593} C_VEL
LIN {X 0,Y 392.462,Z 716.956,A -85,B 0,C 180,E1 -11773.752,E2 -11773.752} C_VEL
LIN {X 0,Y 391.509,Z 727.29,A -85,B 0,C 180,E1 -11775.179,E2 -11775.179} C_VEL
LIN {X 0,Y 390.826,Z 734.896,A -85,B 0,C 180,E1 -11776.481,E2 -11776.481} C_VEL
LIN {X 0,Y 390.208,Z 742.312,A -85,B 0,C 180,E1 -11778.046,E2 -11778.046} C_VEL
LIN {X 0,Y 389.589,Z 748.27,A -85,B 0,C 180,E1 -11779.607,E2 -11779.607} C_VEL
LIN {X 0,Y 389.197,Z 752.971,A -85,B 0,C 180,E1 -11781.171,E2 -11781.171} C_VEL
LIN {X 0,Y 388.939,Z 756.556,A -85,B 0,C 180,E1 -11782.734,E2 -11782.734} C_VEL
LIN {X 0,Y 388.837,Z 758.401,A -85,B 0,C 180,E1 -11783.774,E2 -11783.774} C_VEL
LIN {X 0,Y 388.781,Z 759.791,A -85,B 0,C 180,E1 -11784.814,E2 -11784.814} C_VEL
LIN {X 0,Y 388.657,Z 761.368,A -85,B 0,C 180,E1 -11786.89,E2 -11786.89} C_VEL
LIN {X 0,Y 388.709,Z 761.578,A -85,B 0,C 180,E1 -11787.928,E2 -11787.928} C_VEL
LIN {X 0,Y 388.71,Z 761.358,A -85,B 0,C 180,E1 -11788.964,E2 -11788.964} C_VEL
LIN {X 0,Y 388.74,Z 759.771,A -85,B 0,C 180,E1 -11791.036,E2 -11791.036} C_VEL
LIN {X 0,Y 388.878,Z 758.373,A -85,B 0,C 180,E1 -11792.071,E2 -11792.071} C_VEL
LIN {X 0,Y 389.083,Z 755.471,A -85,B 0,C 180,E1 -11793.625,E2 -11793.625} C_VEL
LIN {X 0,Y 389.198,Z 751.542,A -85,B 0,C 180,E1 -11795.18,E2 -11795.18} C_VEL
LIN {X 0,Y 389.388,Z 749.468,A -85,B 0,C 180,E1 -11795.85,E2 -11795.85} C_VEL
LIN {X 0,Y 388.976,Z 746.912,A -85,B 0,C 180,E1 -11796.628,E2 -11796.628} C_VEL
LIN {X 0,Y 386.533,Z 742.321,A -85,B 0,C 180,E1 -11797.881,E2 -11797.881} C_VEL
LIN {X 0,Y 384.118,Z 737.18,A -85,B 0,C 180,E1 -11799.094,E2 -11799.094} C_VEL
LIN {X 0,Y 383.752,Z 733.621,A -85,B 0,C 180,E1 -11799.798,E2 -11799.798} C_VEL
LIN {X 0,Y 384.664,Z 724.316,A -85,B 0,C 180,E1 -11801.327,E2 -11801.327} C_VEL
LIN {X 0,Y 385.535,Z 714.364,A -85,B 0,C 180,E1 -11802.635,E2 -11802.635} C_VEL
LIN {X 0,Y 386.433,Z 703.199,A -85,B 0,C 180,E1 -11803.81,E2 -11803.81} C_VEL
LIN {X 0,Y 387.211,Z 692.248,A -85,B 0,C 180,E1 -11804.72,E2 -11804.72} C_VEL
LIN {X 0,Y 388.047,Z 679.91,A -85,B 0,C 180,E1 -11805.494,E2 -11805.494} C_VEL
LIN {X 0,Y 388.506,Z 667.463,A -85,B 0,C 180,E1 -11806.066,E2 -11806.066} C_VEL
LIN {X 0,Y 388.863,Z 654.093,A -85,B 0,C 180,E1 -11806.454,E2 -11806.454} C_VEL
LIN {X 0,Y 389.942,Z 571.778,A -85,B 0,C 180,E1 -11807.977,E2 -11807.977} C_VEL
LIN {X 0,Y 385.839,Z 548.57,A -85,B 0,C 180,E1 -11808.649,E2 -11808.649} C_VEL
LIN {X 0,Y 386.625,Z 531.138,A -85,B 0,C 180,E1 -11811.843,E2 -11811.843} C_VEL
LIN {X 0,Y 386.422,Z 528.054,A -85,B 0,C 180,E1 -11812.453,E2 -11812.453} C_VEL
LIN {X 0,Y 384.028,Z 516.142,A -85,B 0,C 180,E1 -11814.892,E2 -11814.892} C_VEL
LIN {X 0,Y 383.081,Z 511.77,A -85,B 0,C 180,E1 -11815.866,E2 -11815.866} C_VEL
LIN {X 0,Y 383.042,Z 511.774,A -85,B 0,C 180,E1 -11818.492,E2 -11818.492} C_VEL
LIN {X 0,Y 383.01,Z 511.777,A -85,B 0,C 180,E1 -11822.149,E2 -11822.149} C_VEL
LIN {X 0,Y 383.018,Z 511.774,A -85,B 0,C 180,E1 -11824.667,E2 -11824.667} C_VEL
LIN {X 0,Y 382.999,Z 511.775,A -85,B 0,C 180,E1 -11827.903,E2 -11827.903} C_VEL
LIN {X 0,Y 383.041,Z 511.771,A -85,B 0,C 180,E1 -11831.339,E2 -11831.339} C_VEL
LIN {X 0,Y 383.033,Z 511.769,A -85,B 0,C 180,E1 -11834.308,E2 -11834.308} C_VEL
LIN {X 0,Y 383.007,Z 511.776,A -85,B 0,C 180,E1 -11837.239,E2 -11837.239} C_VEL
LIN {X 0,Y 383.013,Z 511.776,A -85,B 0,C 180,E1 -11840.412,E2 -11840.412} C_VEL
LIN {X 0,Y 383.035,Z 511.846,A -85,B 0,C 180,E1 -11843.758,E2 -11843.758} C_VEL
LIN {X 0,Y 389.519,Z 529.867,A -85,B 0,C 180,E1 -11844.464,E2 -11844.464} C_VEL
LIN {X 0,Y 387.764,Z 616.415,A -85,B 0,C 180,E1 -11846.359,E2 -11846.359} C_VEL
LIN {X 0,Y 387.381,Z 629.333,A -85,B 0,C 180,E1 -11846.845,E2 -11846.845} C_VEL
LIN {X 0,Y 386.893,Z 641.818,A -85,B 0,C 180,E1 -11847.519,E2 -11847.519} C_VEL
LIN {X 0,Y 386.183,Z 654.773,A -85,B 0,C 180,E1 -11848.467,E2 -11848.467} C_VEL
LIN {X 0,Y 385.513,Z 665.421,A -85,B 0,C 180,E1 -11849.458,E2 -11849.458} C_VEL
LIN {X 0,Y 384.854,Z 675.33,A -85,B 0,C 180,E1 -11850.597,E2 -11850.597} C_VEL
LIN {X 0,Y 384.177,Z 684.539,A -85,B 0,C 180,E1 -11851.896,E2 -11851.896} C_VEL
LIN {X 0,Y 383.55,Z 692.833,A -85,B 0,C 180,E1 -11853.325,E2 -11853.325} C_VEL
LIN {X 0,Y 383.053,Z 699.606,A -85,B 0,C 180,E1 -11854.749,E2 -11854.749} C_VEL
LIN {X 0,Y 382.684,Z 705.128,A -85,B 0,C 180,E1 -11856.169,E2 -11856.169} C_VEL
LIN {X 0,Y 382.331,Z 710.379,A -85,B 0,C 180,E1 -11857.862,E2 -11857.862} C_VEL
LIN {X 0,Y 382.041,Z 714.655,A -85,B 0,C 180,E1 -11859.746,E2 -11859.746} C_VEL
LIN {X 0,Y 381.852,Z 717.65,A -85,B 0,C 180,E1 -11861.766,E2 -11861.766} C_VEL
LIN {X 0,Y 381.836,Z 718.784,A -85,B 0,C 180,E1 -11863.152,E2 -11863.152} C_VEL
LIN {X 0,Y 381.846,Z 719.197,A -85,B 0,C 180,E1 -11865.068,E2 -11865.068} C_VEL
LIN {X 0,Y 381.918,Z 718.823,A -85,B 0,C 180,E1 -11866.159,E2 -11866.159} C_VEL
LIN {X 0,Y 382.033,Z 717.97,A -85,B 0,C 180,E1 -11867.246,E2 -11867.246} C_VEL
LIN {X 0,Y 382.18,Z 716.701,A -85,B 0,C 180,E1 -11868.329,E2 -11868.329} C_VEL
LIN {X 0,Y 382.511,Z 713.926,A -85,B 0,C 180,E1 -11869.947,E2 -11869.947} C_VEL
LIN {X 0,Y 382.946,Z 710.068,A -85,B 0,C 180,E1 -11871.557,E2 -11871.557} C_VEL
LIN {X 0,Y 383.515,Z 705.046,A -85,B 0,C 180,E1 -11873.159,E2 -11873.159} C_VEL
LIN {X 0,Y 384.179,Z 698.696,A -85,B 0,C 180,E1 -11874.752,E2 -11874.752} C_VEL
LIN {X 0,Y 384.999,Z 690.753,A -85,B 0,C 180,E1 -11876.337,E2 -11876.337} C_VEL
LIN {X 0,Y 385.822,Z 682.642,A -85,B 0,C 180,E1 -11877.651,E2 -11877.651} C_VEL
LIN {X 0,Y 386.703,Z 672.772,A -85,B 0,C 180,E1 -11878.958,E2 -11878.958} C_VEL
LIN {X 0,Y 387.71,Z 661.584,A -85,B 0,C 180,E1 -11880.13,E2 -11880.13} C_VEL
LIN {X 0,Y 388.528,Z 650.727,A -85,B 0,C 180,E1 -11881.036,E2 -11881.036} C_VEL
LIN {X 0,Y 389.197,Z 638.854,A -85,B 0,C 180,E1 -11881.811,E2 -11881.811} C_VEL
LIN {X 0,Y 389.755,Z 625.239,A -85,B 0,C 180,E1 -11882.454,E2 -11882.454} C_VEL
LIN {X 0,Y 390.1,Z 611.477,A -85,B 0,C 180,E1 -11882.872,E2 -11882.872} C_VEL
LIN {X 0,Y 392.411,Z 533.256,A -85,B 0,C 180,E1 -11884.694,E2 -11884.694} C_VEL
LIN {X 0,Y 383.802,Z 514.072,A -85,B 0,C 180,E1 -11885.911,E2 -11885.911} C_VEL
LIN {X 0,Y 383.278,Z 511.745,A -85,B 0,C 180,E1 -11886.779,E2 -11886.779} C_VEL
LIN {X 0,Y 383.148,Z 511.761,A -85,B 0,C 180,E1 -11889.502,E2 -11889.502} C_VEL
LIN {X 0,Y 383.134,Z 511.761,A -85,B 0,C 180,E1 -11892.716,E2 -11892.716} C_VEL
LIN {X 0,Y 383.073,Z 511.768,A -85,B 0,C 180,E1 -11895.974,E2 -11895.974} C_VEL
LIN {X 0,Y 383.052,Z 511.772,A -85,B 0,C 180,E1 -11899.284,E2 -11899.284} C_VEL
LIN {X 0,Y 383.03,Z 511.772,A -85,B 0,C 180,E1 -11903.451,E2 -11903.451} C_VEL
LIN {X 0,Y 383.073,Z 511.764,A -85,B 0,C 180,E1 -11906.124,E2 -11906.124} C_VEL
LIN {X 0,Y 383.043,Z 511.767,A -85,B 0,C 180,E1 -11908.492,E2 -11908.492} C_VEL
LIN {X 0,Y 383.004,Z 511.77,A -85,B 0,C 180,E1 -11912.15,E2 -11912.15} C_VEL
LIN {X 0,Y 383.012,Z 511.772,A -85,B 0,C 180,E1 -11914.668,E2 -11914.668} C_VEL
LIN {X 0,Y 382.996,Z 511.774,A -85,B 0,C 180,E1 -11917.905,E2 -11917.905} C_VEL
LIN {X 0,Y 382.979,Z 511.78,A -85,B 0,C 180,E1 -11921.348,E2 -11921.348} C_VEL
LIN {X 0,Y 382.992,Z 511.777,A -85,B 0,C 180,E1 -11924.304,E2 -11924.304} C_VEL
LIN {X 0,Y 383.006,Z 511.778,A -85,B 0,C 180,E1 -11927.241,E2 -11927.241} C_VEL
LIN {X 0,Y 383.013,Z 511.777,A -85,B 0,C 180,E1 -11930.414,E2 -11930.414} C_VEL
LIN {X 0,Y 383.024,Z 511.774,A -85,B 0,C 180,E1 -11934.045,E2 -11934.045} C_VEL
LIN {X 0,Y 383.015,Z 511.848,A -85,B 0,C 180,E1 -11937.272,E2 -11937.272} C_VEL
LIN {X 0,Y 385.546,Z 521.735,A -85,B 0,C 180,E1 -11939.915,E2 -11939.915} C_VEL
LIN {X 0,Y 387.499,Z 530.689,A -85,B 0,C 180,E1 -11942.122,E2 -11942.122} C_VEL
LIN {X 0,Y 388.103,Z 534.864,A -85,B 0,C 180,E1 -11943.083,E2 -11943.083} C_VEL
LIN {X 0,Y 386.355,Z 552.57,A -85,B 0,C 180,E1 -11946.694,E2 -11946.694} C_VEL
LIN {X 0,Y 385.622,Z 560.396,A -85,B 0,C 180,E1 -11948.244,E2 -11948.244} C_VEL
LIN {X 0,Y 389.057,Z 580.625,A -85,B 0,C 180,E1 -11949.031,E2 -11949.031} C_VEL
LIN {X 0,Y 391.122,Z 600.069,A -85,B 0,C 180,E1 -11949.676,E2 -11949.676} C_VEL
LIN {X 0,Y 389.121,Z 672.918,A -85,B 0,C 180,E1 -11951.37,E2 -11951.37} C_VEL
LIN {X 0,Y 388.395,Z 686.283,A -85,B 0,C 180,E1 -11951.881,E2 -11951.881} C_VEL
LIN {X 0,Y 387.39,Z 699.101,A -85,B 0,C 180,E1 -11952.582,E2 -11952.582} C_VEL
LIN {X 0,Y 386.143,Z 716.29,A -85,B 0,C 180,E1 -11953.75,E2 -11953.75} C_VEL
LIN {X 0,Y 385.241,Z 727.98,A -85,B 0,C 180,E1 -11954.797,E2 -11954.797} C_VEL
LIN {X 0,Y 384.376,Z 739.295,A -85,B 0,C 180,E1 -11956.088,E2 -11956.088} C_VEL
LIN {X 0,Y 383.645,Z 747.854,A -85,B 0,C 180,E1 -11957.301,E2 -11957.301} C_VEL
LIN {X 0,Y 382.836,Z 756.896,A -85,B 0,C 180,E1 -11958.887,E2 -11958.887} C_VEL
LIN {X 0,Y 382.309,Z 764.162,A -85,B 0,C 180,E1 -11960.477,E2 -11960.477} C_VEL
LIN {X 0,Y 381.949,Z 769.951,A -85,B 0,C 180,E1 -11962.068,E2 -11962.068} C_VEL
LIN {X 0,Y 381.757,Z 774.778,A -85,B 0,C 180,E1 -11963.785,E2 -11963.785} C_VEL
LIN {X 0,Y 381.654,Z 778.801,A -85,B 0,C 180,E1 -11965.776,E2 -11965.776} C_VEL
LIN {X 0,Y 381.603,Z 780.314,A -85,B 0,C 180,E1 -11966.833,E2 -11966.833} C_VEL
LIN {X 0,Y 381.634,Z 781.369,A -85,B 0,C 180,E1 -11967.889,E2 -11967.889} C_VEL
LIN {X 0,Y 381.648,Z 782.027,A -85,B 0,C 180,E1 -11968.945,E2 -11968.945} C_VEL
LIN {X 0,Y 381.647,Z 782.294,A -85,B 0,C 180,E1 -11970,E2 -11970} C_VEL
LIN {X 0,Y 381.631,Z 782.147,A -85,B 0,C 180,E1 -11971.055,E2 -11971.055} C_VEL
LIN {X 0,Y 381.633,Z 781.569,A -85,B 0,C 180,E1 -11972.111,E2 -11972.111} C_VEL
LIN {X 0,Y 381.655,Z 779.233,A -85,B 0,C 180,E1 -11974.224,E2 -11974.224} C_VEL
LIN {X 0,Y 381.757,Z 775.415,A -85,B 0,C 180,E1 -11976.216,E2 -11976.216} C_VEL
LIN {X 0,Y 381.993,Z 770.804,A -85,B 0,C 180,E1 -11977.931,E2 -11977.931} C_VEL
LIN {X 0,Y 382.358,Z 765.277,A -85,B 0,C 180,E1 -11979.522,E2 -11979.522} C_VEL
LIN {X 0,Y 382.873,Z 758.363,A -85,B 0,C 180,E1 -11981.112,E2 -11981.112} C_VEL
LIN {X 0,Y 383.742,Z 749.681,A -85,B 0,C 180,E1 -11982.695,E2 -11982.695} C_VEL
LIN {X 0,Y 384.606,Z 740.052,A -85,B 0,C 180,E1 -11984.111,E2 -11984.111} C_VEL
LIN {X 0,Y 385.494,Z 729.701,A -85,B 0,C 180,E1 -11985.328,E2 -11985.328} C_VEL
LIN {X 0,Y 386.501,Z 718.479,A -85,B 0,C 180,E1 -11986.37,E2 -11986.37} C_VEL
LIN {X 0,Y 387.371,Z 706.827,A -85,B 0,C 180,E1 -11987.214,E2 -11987.214} C_VEL
LIN {X 0,Y 388.144,Z 694.008,A -85,B 0,C 180,E1 -11987.893,E2 -11987.893} C_VEL
LIN {X 0,Y 388.71,Z 681.421,A -85,B 0,C 180,E1 -11988.343,E2 -11988.343} C_VEL
LIN {X 0,Y 389.196,Z 655.139,A -85,B 0,C 180,E1 -11988.865,E2 -11988.865} C_VEL
LIN {X 0,Y 389.802,Z 597.961,A -85,B 0,C 180,E1 -11989.929,E2 -11989.929} C_VEL
LIN {X 0,Y 385.241,Z 564.522,A -85,B 0,C 180,E1 -11990.838,E2 -11990.838} C_VEL
LIN {X 0,Y 384.957,Z 562.249,A -85,B 0,C 180,E1 -11990.924,E2 -11990.924} C_VEL
LIN {X 0,Y 386.489,Z 542.937,A -85,B 0,C 180,E1 -11994.603,E2 -11994.603} C_VEL
LIN {X 0,Y 387.228,Z 532.112,A -85,B 0,C 180,E1 -11996.692,E2 -11996.692} C_VEL
LIN {X 0,Y 384.916,Z 520.515,A -85,B 0,C 180,E1 -11999.13,E2 -11999.13} C_VEL
LIN {X 0,Y 383.019,Z 511.777,A -85,B 0,C 180,E1 -12001.068,E2 -12001.068} C_VEL
LIN {X 0,Y 383.015,Z 511.775,A -85,B 0,C 180,E1 -12004.667,E2 -12004.667} C_VEL
LIN {X 0,Y 382.997,Z 511.748,A -85,B 0,C 180,E1 -12007.903,E2 -12007.903} C_VEL
LIN {X 0,Y 382.983,Z 511.782,A -85,B 0,C 180,E1 -12011.346,E2 -12011.346} C_VEL
LIN {X 0,Y 382.994,Z 511.771,A -85,B 0,C 180,E1 -12014.303,E2 -12014.303} C_VEL
LIN {X 0,Y 383.035,Z 511.768,A -85,B 0,C 180,E1 -12017.244,E2 -12017.244} C_VEL
LIN {X 0,Y 383.016,Z 511.773,A -85,B 0,C 180,E1 -12020.412,E2 -12020.412} C_VEL
LIN {X 0,Y 383.021,Z 511.765,A -85,B 0,C 180,E1 -12024.044,E2 -12024.044} C_VEL
LIN {X 0,Y 382.981,Z 511.773,A -85,B 0,C 180,E1 -12027.577,E2 -12027.577} C_VEL
LIN {X 0,Y 382.991,Z 511.767,A -85,B 0,C 180,E1 -12030.3,E2 -12030.3} C_VEL
LIN {X 0,Y 383.05,Z 511.77,A -85,B 0,C 180,E1 -12032.698,E2 -12032.698} C_VEL
LIN {X 0,Y 383.043,Z 511.758,A -85,B 0,C 180,E1 -12035.039,E2 -12035.039} C_VEL
LIN {X 0,Y 382.984,Z 511.773,A -85,B 0,C 180,E1 -12038.469,E2 -12038.469} C_VEL
LIN {X 0,Y 383.055,Z 511.759,A -85,B 0,C 180,E1 -12041.826,E2 -12041.826} C_VEL
LIN {X 0,Y 383.103,Z 511.753,A -85,B 0,C 180,E1 -12045.118,E2 -12045.118} C_VEL
LIN {X 0,Y 383.099,Z 511.762,A -85,B 0,C 180,E1 -12048.358,E2 -12048.358} C_VEL
LIN {X 0,Y 383.256,Z 511.724,A -85,B 0,C 180,E1 -12051.974,E2 -12051.974} C_VEL
LIN {X 0,Y 383.198,Z 511.748,A -85,B 0,C 180,E1 -12054.739,E2 -12054.739} C_VEL
LIN {X 0,Y 383.379,Z 511.721,A -85,B 0,C 180,E1 -12057.899,E2 -12057.899} C_VEL
LIN {X 0,Y 383.513,Z 511.688,A -85,B 0,C 180,E1 -12060,E2 -12060} C_VEL
LIN {X 0,Y 383.247,Z 511.745,A -85,B 0,C 180,E1 -12063.154,E2 -12063.154} C_VEL
LIN {X 0,Y 383.261,Z 511.733,A -85,B 0,C 180,E1 -12066.585,E2 -12066.585} C_VEL
LIN {X 0,Y 383.144,Z 511.746,A -85,B 0,C 180,E1 -12069.503,E2 -12069.503} C_VEL
LIN {X 0,Y 383.118,Z 511.758,A -85,B 0,C 180,E1 -12073.537,E2 -12073.537} C_VEL
LIN {X 0,Y 383.087,Z 511.756,A -85,B 0,C 180,E1 -12077.455,E2 -12077.455} C_VEL
LIN {X 0,Y 383.022,Z 511.774,A -85,B 0,C 180,E1 -12080.648,E2 -12080.648} C_VEL
LIN {X 0,Y 383.027,Z 511.761,A -85,B 0,C 180,E1 -12083.808,E2 -12083.808} C_VEL
LIN {X 0,Y 383.074,Z 511.765,A -85,B 0,C 180,E1 -12086.124,E2 -12086.124} C_VEL
LIN {X 0,Y 383.044,Z 511.767,A -85,B 0,C 180,E1 -12088.493,E2 -12088.493} C_VEL
LIN {X 0,Y 383.004,Z 511.775,A -85,B 0,C 180,E1 -12092.428,E2 -12092.428} C_VEL
LIN {X 0,Y 383.03,Z 511.77,A -85,B 0,C 180,E1 -12096.166,E2 -12096.166} C_VEL
LIN {X 0,Y 383.006,Z 511.772,A -85,B 0,C 180,E1 -12099.959,E2 -12099.959} C_VEL
LIN {X 0,Y 383.003,Z 511.778,A -85,B 0,C 180,E1 -12102.78,E2 -12102.78} C_VEL
LIN {X 0,Y 382.999,Z 511.777,A -85,B 0,C 180,E1 -12105.791,E2 -12105.791} C_VEL
LIN {X 0,Y 382.988,Z 511.78,A -85,B 0,C 180,E1 -12108.797,E2 -12108.797} C_VEL
LIN {X 0,Y 382.999,Z 511.773,A -85,B 0,C 180,E1 -12112.097,E2 -12112.097} C_VEL
LIN {X 0,Y 383.018,Z 511.767,A -85,B 0,C 180,E1 -12115.333,E2 -12115.333} C_VEL
LIN {X 0,Y 382.984,Z 511.781,A -85,B 0,C 180,E1 -12119.082,E2 -12119.082} C_VEL
LIN {X 0,Y 383.023,Z 511.882,A -85,B 0,C 180,E1 -12119.797,E2 -12119.797} C_VEL
LIN {X 0,Y 385.748,Z 523.608,A -85,B 0,C 180,E1 -12122.317,E2 -12122.317} C_VEL
LIN {X 0,Y 387.067,Z 531.183,A -85,B 0,C 180,E1 -12123.878,E2 -12123.878} C_VEL
LIN {X 0,Y 386.421,Z 544.85,A -85,B 0,C 180,E1 -12126.415,E2 -12126.415} C_VEL
LIN {X 0,Y 386.314,Z 548.859,A -85,B 0,C 180,E1 -12127.096,E2 -12127.096} C_VEL
LIN {X 0,Y 390.785,Z 572.226,A -85,B 0,C 180,E1 -12127.811,E2 -12127.811} C_VEL
LIN {X 0,Y 389.439,Z 658.478,A -85,B 0,C 180,E1 -12129.431,E2 -12129.431} C_VEL
LIN {X 0,Y 388.98,Z 671.114,A -85,B 0,C 180,E1 -12129.854,E2 -12129.854} C_VEL
LIN {X 0,Y 388.402,Z 683.895,A -85,B 0,C 180,E1 -12130.511,E2 -12130.511} C_VEL
LIN {X 0,Y 387.593,Z 696.128,A -85,B 0,C 180,E1 -12131.363,E2 -12131.363} C_VEL
LIN {X 0,Y 386.604,Z 707.682,A -85,B 0,C 180,E1 -12132.409,E2 -12132.409} C_VEL
LIN {X 0,Y 385.54,Z 718.004,A -85,B 0,C 180,E1 -12133.588,E2 -12133.588} C_VEL
LIN {X 0,Y 384.616,Z 727.33,A -85,B 0,C 180,E1 -12134.907,E2 -12134.907} C_VEL
LIN {X 0,Y 383.897,Z 734.967,A -85,B 0,C 180,E1 -12136.232,E2 -12136.232} C_VEL
LIN {X 0,Y 383.244,Z 742.409,A -85,B 0,C 180,E1 -12137.826,E2 -12137.826} C_VEL
LIN {X 0,Y 382.556,Z 748.385,A -85,B 0,C 180,E1 -12139.414,E2 -12139.414} C_VEL
LIN {X 0,Y 382.154,Z 753.102,A -85,B 0,C 180,E1 -12141.007,E2 -12141.007} C_VEL
LIN {X 0,Y 381.868,Z 756.703,A -85,B 0,C 180,E1 -12142.598,E2 -12142.598} C_VEL
LIN {X 0,Y 381.763,Z 758.743,A -85,B 0,C 180,E1 -12143.78,E2 -12143.78} C_VEL
LIN {X 0,Y 381.623,Z 760.945,A -85,B 0,C 180,E1 -12145.776,E2 -12145.776} C_VEL
LIN {X 0,Y 381.607,Z 761.769,A -85,B 0,C 180,E1 -12147.889,E2 -12147.889} C_VEL
LIN {X 0,Y 381.625,Z 761.558,A -85,B 0,C 180,E1 -12148.945,E2 -12148.945} C_VEL
LIN {X 0,Y 381.656,Z 759.985,A -85,B 0,C 180,E1 -12151.055,E2 -12151.055} C_VEL
LIN {X 0,Y 381.797,Z 758.6,A -85,B 0,C 180,E1 -12152.11,E2 -12152.11} C_VEL
LIN {X 0,Y 382.005,Z 755.71,A -85,B 0,C 180,E1 -12153.692,E2 -12153.692} C_VEL
LIN {X 0,Y 382.146,Z 751.795,A -85,B 0,C 180,E1 -12155.276,E2 -12155.276} C_VEL
LIN {X 0,Y 382.659,Z 746.064,A -85,B 0,C 180,E1 -12157.035,E2 -12157.035} C_VEL
LIN {X 0,Y 383.243,Z 739.152,A -85,B 0,C 180,E1 -12158.702,E2 -12158.702} C_VEL
LIN {X 0,Y 383.752,Z 733.621,A -85,B 0,C 180,E1 -12159.798,E2 -12159.798} C_VEL
LIN {X 0,Y 383.419,Z 729.896,A -85,B 0,C 180,E1 -12160.478,E2 -12160.478} C_VEL
LIN {X 0,Y 381.193,Z 723.55,A -85,B 0,C 180,E1 -12161.571,E2 -12161.571} C_VEL
LIN {X 0,Y 379.052,Z 716.702,A -85,B 0,C 180,E1 -12162.603,E2 -12162.603} C_VEL
LIN {X 0,Y 378.85,Z 712.133,A -85,B 0,C 180,E1 -12163.175,E2 -12163.175} C_VEL
LIN {X 0,Y 379.713,Z 702.224,A -85,B 0,C 180,E1 -12164.196,E2 -12164.196} C_VEL
LIN {X 0,Y 380.529,Z 690.86,A -85,B 0,C 180,E1 -12165.122,E2 -12165.122} C_VEL
LIN {X 0,Y 381.367,Z 678.039,A -85,B 0,C 180,E1 -12165.909,E2 -12165.909} C_VEL
LIN {X 0,Y 381.799,Z 665.55,A -85,B 0,C 180,E1 -12166.458,E2 -12166.458} C_VEL
LIN {X 0,Y 382.153,Z 652.385,A -85,B 0,C 180,E1 -12166.811,E2 -12166.811} C_VEL
LIN {X 0,Y 383.302,Z 572.991,A -85,B 0,C 180,E1 -12168.3,E2 -12168.3} C_VEL
LIN {X 0,Y 379.01,Z 548.678,A -85,B 0,C 180,E1 -12169.027,E2 -12169.027} C_VEL
LIN {X 0,Y 379.771,Z 532.04,A -85,B 0,C 180,E1 -12172.093,E2 -12172.093} C_VEL
LIN {X 0,Y 378.684,Z 525.133,A -85,B 0,C 180,E1 -12173.516,E2 -12173.516} C_VEL
LIN {X 0,Y 376.035,Z 512.648,A -85,B 0,C 180,E1 -12176.148,E2 -12176.148} C_VEL
LIN {X 0,Y 375.972,Z 512.654,A -85,B 0,C 180,E1 -12179.078,E2 -12179.078} C_VEL
LIN {X 0,Y 375.95,Z 512.658,A -85,B 0,C 180,E1 -12182.828,E2 -12182.828} C_VEL
LIN {X 0,Y 375.957,Z 512.653,A -85,B 0,C 180,E1 -12185.415,E2 -12185.415} C_VEL
LIN {X 0,Y 375.973,Z 512.651,A -85,B 0,C 180,E1 -12188.269,E2 -12188.269} C_VEL
LIN {X 0,Y 375.985,Z 512.649,A -85,B 0,C 180,E1 -12191.609,E2 -12191.609} C_VEL
LIN {X 0,Y 375.968,Z 512.642,A -85,B 0,C 180,E1 -12195.261,E2 -12195.261} C_VEL
LIN {X 0,Y 375.938,Z 512.658,A -85,B 0,C 180,E1 -12199.132,E2 -12199.132} C_VEL
LIN {X 0,Y 375.962,Z 512.653,A -85,B 0,C 180,E1 -12201.911,E2 -12201.911} C_VEL
LIN {X 0,Y 375.978,Z 512.678,A -85,B 0,C 180,E1 -12203.45,E2 -12203.45} C_VEL
LIN {X 0,Y 382.678,Z 531.859,A -85,B 0,C 180,E1 -12204.209,E2 -12204.209} C_VEL
LIN {X 0,Y 380.875,Z 616.816,A -85,B 0,C 180,E1 -12206.119,E2 -12206.119} C_VEL
LIN {X 0,Y 380.447,Z 630.795,A -85,B 0,C 180,E1 -12206.662,E2 -12206.662} C_VEL
LIN {X 0,Y 379.906,Z 643.704,A -85,B 0,C 180,E1 -12207.398,E2 -12207.398} C_VEL
LIN {X 0,Y 379.24,Z 655.361,A -85,B 0,C 180,E1 -12208.276,E2 -12208.276} C_VEL
LIN {X 0,Y 378.546,Z 666.133,A -85,B 0,C 180,E1 -12209.298,E2 -12209.298} C_VEL
LIN {X 0,Y 377.828,Z 676.52,A -85,B 0,C 180,E1 -12210.528,E2 -12210.528} C_VEL
LIN {X 0,Y 377.058,Z 686.092,A -85,B 0,C 180,E1 -12211.924,E2 -12211.924} C_VEL
LIN {X 0,Y 376.464,Z 694.241,A -85,B 0,C 180,E1 -12213.381,E2 -12213.381} C_VEL
LIN {X 0,Y 375.946,Z 700.871,A -85,B 0,C 180,E1 -12214.83,E2 -12214.83} C_VEL
LIN {X 0,Y 375.529,Z 706.979,A -85,B 0,C 180,E1 -12216.493,E2 -12216.493} C_VEL
LIN {X 0,Y 375.235,Z 711.373,A -85,B 0,C 180,E1 -12218,E2 -12218} C_VEL
LIN {X 0,Y 374.988,Z 714.889,A -85,B 0,C 180,E1 -12219.566,E2 -12219.566} C_VEL
LIN {X 0,Y 374.796,Z 717.759,A -85,B 0,C 180,E1 -12221.411,E2 -12221.411} C_VEL
LIN {X 0,Y 374.763,Z 719.245,A -85,B 0,C 180,E1 -12223.016,E2 -12223.016} C_VEL
LIN {X 0,Y 374.758,Z 719.792,A -85,B 0,C 180,E1 -12224.778,E2 -12224.778} C_VEL
LIN {X 0,Y 374.827,Z 719.559,A -85,B 0,C 180,E1 -12225.892,E2 -12225.892} C_VEL
LIN {X 0,Y 374.956,Z 718.845,A -85,B 0,C 180,E1 -12227.069,E2 -12227.069} C_VEL
LIN {X 0,Y 375.088,Z 717.762,A -85,B 0,C 180,E1 -12228.105,E2 -12228.105} C_VEL
LIN {X 0,Y 375.436,Z 715.23,A -85,B 0,C 180,E1 -12229.756,E2 -12229.756} C_VEL
LIN {X 0,Y 375.881,Z 711.631,A -85,B 0,C 180,E1 -12231.397,E2 -12231.397} C_VEL
LIN {X 0,Y 376.449,Z 706.882,A -85,B 0,C 180,E1 -12233.03,E2 -12233.03} C_VEL
LIN {X 0,Y 377.096,Z 700.866,A -85,B 0,C 180,E1 -12234.653,E2 -12234.653} C_VEL
LIN {X 0,Y 377.978,Z 693.33,A -85,B 0,C 180,E1 -12236.268,E2 -12236.268} C_VEL
LIN {X 0,Y 378.766,Z 685.626,A -85,B 0,C 180,E1 -12237.607,E2 -12237.607} C_VEL
LIN {X 0,Y 379.725,Z 676.206,A -85,B 0,C 180,E1 -12238.939,E2 -12238.939} C_VEL
LIN {X 0,Y 380.743,Z 665.839,A -85,B 0,C 180,E1 -12240.132,E2 -12240.132} C_VEL
LIN {X 0,Y 381.698,Z 654.318,A -85,B 0,C 180,E1 -12241.187,E2 -12241.187} C_VEL
LIN {X 0,Y 382.588,Z 641.172,A -85,B 0,C 180,E1 -12242.105,E2 -12242.105} C_VEL
LIN {X 0,Y 383.166,Z 628.388,A -85,B 0,C 180,E1 -12242.759,E2 -12242.759} C_VEL
LIN {X 0,Y 383.582,Z 614.862,A -85,B 0,C 180,E1 -12243.216,E2 -12243.216} C_VEL
LIN {X 0,Y 386.058,Z 535.166,A -85,B 0,C 180,E1 -12245.132,E2 -12245.132} C_VEL
LIN {X 0,Y 377.983,Z 517.546,A -85,B 0,C 180,E1 -12246.306,E2 -12246.306} C_VEL
LIN {X 0,Y 376.76,Z 514.941,A -85,B 0,C 180,E1 -12246.493,E2 -12246.493} C_VEL
LIN {X 0,Y 376.239,Z 512.621,A -85,B 0,C 180,E1 -12247.378,E2 -12247.378} C_VEL
LIN {X 0,Y 376.085,Z 512.641,A -85,B 0,C 180,E1 -12250.77,E2 -12250.77} C_VEL
LIN {X 0,Y 376.058,Z 512.643,A -85,B 0,C 180,E1 -12254.061,E2 -12254.061} C_VEL
LIN {X 0,Y 376.035,Z 512.645,A -85,B 0,C 180,E1 -12257.607,E2 -12257.607} C_VEL
LIN {X 0,Y 375.971,Z 512.654,A -85,B 0,C 180,E1 -12260.832,E2 -12260.832} C_VEL
LIN {X 0,Y 375.986,Z 512.648,A -85,B 0,C 180,E1 -12264.282,E2 -12264.282} C_VEL
LIN {X 0,Y 376.013,Z 512.645,A -85,B 0,C 180,E1 -12266.653,E2 -12266.653} C_VEL
LIN {X 0,Y 375.97,Z 512.65,A -85,B 0,C 180,E1 -12269.079,E2 -12269.079} C_VEL
LIN {X 0,Y 375.943,Z 512.654,A -85,B 0,C 180,E1 -12272.829,E2 -12272.829} C_VEL
LIN {X 0,Y 375.952,Z 512.652,A -85,B 0,C 180,E1 -12275.416,E2 -12275.416} C_VEL
LIN {X 0,Y 375.97,Z 512.649,A -85,B 0,C 180,E1 -12278.271,E2 -12278.271} C_VEL
LIN {X 0,Y 375.929,Z 512.656,A -85,B 0,C 180,E1 -12281.601,E2 -12281.601} C_VEL
LIN {X 0,Y 375.95,Z 512.656,A -85,B 0,C 180,E1 -12285.265,E2 -12285.265} C_VEL
LIN {X 0,Y 375.937,Z 512.659,A -85,B 0,C 180,E1 -12289.134,E2 -12289.134} C_VEL
LIN {X 0,Y 375.963,Z 512.654,A -85,B 0,C 180,E1 -12291.912,E2 -12291.912} C_VEL
LIN {X 0,Y 375.978,Z 512.655,A -85,B 0,C 180,E1 -12295.333,E2 -12295.333} C_VEL
LIN {X 0,Y 375.97,Z 512.752,A -85,B 0,C 180,E1 -12296.656,E2 -12296.656} C_VEL
LIN {X 0,Y 378.754,Z 523.479,A -85,B 0,C 180,E1 -12299.658,E2 -12299.658} C_VEL
LIN {X 0,Y 380.67,Z 532.38,A -85,B 0,C 180,E1 -12301.912,E2 -12301.912} C_VEL
LIN {X 0,Y 381.296,Z 536.353,A -85,B 0,C 180,E1 -12302.859,E2 -12302.859} C_VEL
LIN {X 0,Y 379.746,Z 551.211,A -85,B 0,C 180,E1 -12305.974,E2 -12305.974} C_VEL
LIN {X 0,Y 378.895,Z 559.898,A -85,B 0,C 180,E1 -12307.693,E2 -12307.693} C_VEL
LIN {X 0,Y 381.975,Z 576.883,A -85,B 0,C 180,E1 -12308.409,E2 -12308.409} C_VEL
LIN {X 0,Y 384.273,Z 595.836,A -85,B 0,C 180,E1 -12309.09,E2 -12309.09} C_VEL
LIN {X 0,Y 384.621,Z 602.107,A -85,B 0,C 180,E1 -12309.28,E2 -12309.28} C_VEL
LIN {X 0,Y 382.598,Z 671.573,A -85,B 0,C 180,E1 -12310.936,E2 -12310.936} C_VEL
LIN {X 0,Y 381.775,Z 685.727,A -85,B 0,C 180,E1 -12311.486,E2 -12311.486} C_VEL
LIN {X 0,Y 380.833,Z 697.467,A -85,B 0,C 180,E1 -12312.134,E2 -12312.134} C_VEL
LIN {X 0,Y 379.183,Z 717.543,A -85,B 0,C 180,E1 -12313.582,E2 -12313.582} C_VEL
LIN {X 0,Y 378.252,Z 728.945,A -85,B 0,C 180,E1 -12314.647,E2 -12314.647} C_VEL
LIN {X 0,Y 377.51,Z 738.631,A -85,B 0,C 180,E1 -12315.782,E2 -12315.782} C_VEL
LIN {X 0,Y 376.679,Z 747.577,A -85,B 0,C 180,E1 -12317.063,E2 -12317.063} C_VEL
LIN {X 0,Y 375.837,Z 756.634,A -85,B 0,C 180,E1 -12318.677,E2 -12318.677} C_VEL
LIN {X 0,Y 375.253,Z 763.911,A -85,B 0,C 180,E1 -12320.296,E2 -12320.296} C_VEL
LIN {X 0,Y 374.886,Z 769.715,A -85,B 0,C 180,E1 -12321.917,E2 -12321.917} C_VEL
LIN {X 0,Y 374.66,Z 774.914,A -85,B 0,C 180,E1 -12323.823,E2 -12323.823} C_VEL
LIN {X 0,Y 374.579,Z 778.586,A -85,B 0,C 180,E1 -12325.696,E2 -12325.696} C_VEL
LIN {X 0,Y 374.514,Z 780.107,A -85,B 0,C 180,E1 -12326.773,E2 -12326.773} C_VEL
LIN {X 0,Y 374.532,Z 781.167,A -85,B 0,C 180,E1 -12327.849,E2 -12327.849} C_VEL
LIN {X 0,Y 374.549,Z 781.829,A -85,B 0,C 180,E1 -12328.925,E2 -12328.925} C_VEL
LIN {X 0,Y 374.562,Z 782.101,A -85,B 0,C 180,E1 -12330,E2 -12330} C_VEL
LIN {X 0,Y 374.533,Z 781.962,A -85,B 0,C 180,E1 -12331.075,E2 -12331.075} C_VEL
LIN {X 0,Y 374.531,Z 781.389,A -85,B 0,C 180,E1 -12332.151,E2 -12332.151} C_VEL
LIN {X 0,Y 374.581,Z 779.062,A -85,B 0,C 180,E1 -12334.304,E2 -12334.304} C_VEL
LIN {X 0,Y 374.667,Z 775.597,A -85,B 0,C 180,E1 -12336.187,E2 -12336.187} C_VEL
LIN {X 0,Y 374.92,Z 770.657,A -85,B 0,C 180,E1 -12338.082,E2 -12338.082} C_VEL
LIN {X 0,Y 375.332,Z 765.143,A -85,B 0,C 180,E1 -12339.702,E2 -12339.702} C_VEL
LIN {X 0,Y 375.89,Z 758.246,A -85,B 0,C 180,E1 -12341.321,E2 -12341.321} C_VEL
LIN {X 0,Y 376.808,Z 749.585,A -85,B 0,C 180,E1 -12342.933,E2 -12342.933} C_VEL
LIN {X 0,Y 377.679,Z 740.328,A -85,B 0,C 180,E1 -12344.325,E2 -12344.325} C_VEL
LIN {X 0,Y 378.654,Z 729.664,A -85,B 0,C 180,E1 -12345.612,E2 -12345.612} C_VEL
LIN {X 0,Y 379.683,Z 718.48,A -85,B 0,C 180,E1 -12346.672,E2 -12346.672} C_VEL
LIN {X 0,Y 380.611,Z 706.881,A -85,B 0,C 180,E1 -12347.53,E2 -12347.53} C_VEL
LIN {X 0,Y 381.412,Z 694.194,A -85,B 0,C 180,E1 -12348.22,E2 -12348.22} C_VEL
LIN {X 0,Y 382.03,Z 680.688,A -85,B 0,C 180,E1 -12348.71,E2 -12348.71} C_VEL
LIN {X 0,Y 382.606,Z 648.985,A -85,B 0,C 180,E1 -12349.337,E2 -12349.337} C_VEL
LIN {X 0,Y 383.193,Z 598.893,A -85,B 0,C 180,E1 -12350.283,E2 -12350.283} C_VEL
LIN {X 0,Y 378.484,Z 564.186,A -85,B 0,C 180,E1 -12351.25,E2 -12351.25} C_VEL
LIN {X 0,Y 378.046,Z 561.221,A -85,B 0,C 180,E1 -12351.361,E2 -12351.361} C_VEL
LIN {X 0,Y 379.572,Z 543.123,A -85,B 0,C 180,E1 -12354.87,E2 -12354.87} C_VEL
LIN {X 0,Y 380.284,Z 534.236,A -85,B 0,C 180,E1 -12356.614,E2 -12356.614} C_VEL
LIN {X 0,Y 379.017,Z 526.649,A -85,B 0,C 180,E1 -12358.218,E2 -12358.218} C_VEL
LIN {X 0,Y 375.971,Z 512.655,A -85,B 0,C 180,E1 -12361.339,E2 -12361.339} C_VEL
LIN {X 0,Y 375.977,Z 512.652,A -85,B 0,C 180,E1 -12364.667,E2 -12364.667} C_VEL
LIN {X 0,Y 375.971,Z 512.622,A -85,B 0,C 180,E1 -12368.27,E2 -12368.27} C_VEL
LIN {X 0,Y 375.933,Z 512.659,A -85,B 0,C 180,E1 -12371.6,E2 -12371.6} C_VEL
LIN {X 0,Y 375.95,Z 512.657,A -85,B 0,C 180,E1 -12375.264,E2 -12375.264} C_VEL
LIN {X 0,Y 375.976,Z 512.646,A -85,B 0,C 180,E1 -12379.138,E2 -12379.138} C_VEL
LIN {X 0,Y 375.962,Z 512.649,A -85,B 0,C 180,E1 -12381.911,E2 -12381.911} C_VEL
LIN {X 0,Y 375.974,Z 512.653,A -85,B 0,C 180,E1 -12385.332,E2 -12385.332} C_VEL
LIN {X 0,Y 375.953,Z 512.647,A -85,B 0,C 180,E1 -12388.438,E2 -12388.438} C_VEL
LIN {X 0,Y 375.995,Z 512.646,A -85,B 0,C 180,E1 -12392.141,E2 -12392.141} C_VEL
LIN {X 0,Y 375.999,Z 512.643,A -85,B 0,C 180,E1 -12394.539,E2 -12394.539} C_VEL
LIN {X 0,Y 375.949,Z 512.649,A -85,B 0,C 180,E1 -12398.045,E2 -12398.045} C_VEL
LIN {X 0,Y 376.001,Z 512.64,A -85,B 0,C 180,E1 -12401.473,E2 -12401.473} C_VEL
LIN {X 0,Y 376.051,Z 512.628,A -85,B 0,C 180,E1 -12404.832,E2 -12404.832} C_VEL
LIN {X 0,Y 376.051,Z 512.639,A -85,B 0,C 180,E1 -12408.137,E2 -12408.137} C_VEL
LIN {X 0,Y 376.212,Z 512.601,A -85,B 0,C 180,E1 -12411.917,E2 -12411.917} C_VEL
LIN {X 0,Y 376.17,Z 512.623,A -85,B 0,C 180,E1 -12414.64,E2 -12414.64} C_VEL
LIN {X 0,Y 376.346,Z 512.597,A -85,B 0,C 180,E1 -12417.86,E2 -12417.86} C_VEL
LIN {X 0,Y 376.482,Z 512.563,A -85,B 0,C 180,E1 -12420,E2 -12420} C_VEL
LIN {X 0,Y 376.185,Z 512.626,A -85,B 0,C 180,E1 -12423.213,E2 -12423.213} C_VEL
LIN {X 0,Y 376.227,Z 512.612,A -85,B 0,C 180,E1 -12426.571,E2 -12426.571} C_VEL
LIN {X 0,Y 376.111,Z 512.625,A -85,B 0,C 180,E1 -12429.682,E2 -12429.682} C_VEL
LIN {X 0,Y 376.082,Z 512.633,A -85,B 0,C 180,E1 -12433.658,E2 -12433.658} C_VEL
LIN {X 0,Y 376.036,Z 512.637,A -85,B 0,C 180,E1 -12437.607,E2 -12437.607} C_VEL
LIN {X 0,Y 375.972,Z 512.654,A -85,B 0,C 180,E1 -12440.833,E2 -12440.833} C_VEL
LIN {X 0,Y 375.987,Z 512.638,A -85,B 0,C 180,E1 -12444.282,E2 -12444.282} C_VEL
LIN {X 0,Y 376.014,Z 512.647,A -85,B 0,C 180,E1 -12446.653,E2 -12446.653} C_VEL
LIN {X 0,Y 375.972,Z 512.642,A -85,B 0,C 180,E1 -12449.079,E2 -12449.079} C_VEL
LIN {X 0,Y 375.952,Z 512.657,A -85,B 0,C 180,E1 -12452.829,E2 -12452.829} C_VEL
LIN {X 0,Y 375.954,Z 512.649,A -85,B 0,C 180,E1 -12455.416,E2 -12455.416} C_VEL
LIN {X 0,Y 375.972,Z 512.653,A -85,B 0,C 180,E1 -12458.272,E2 -12458.272} C_VEL
LIN {X 0,Y 375.932,Z 512.66,A -85,B 0,C 180,E1 -12461.602,E2 -12461.602} C_VEL
LIN {X 0,Y 375.954,Z 512.658,A -85,B 0,C 180,E1 -12465.265,E2 -12465.265} C_VEL
LIN {X 0,Y 375.94,Z 512.655,A -85,B 0,C 180,E1 -12469.134,E2 -12469.134} C_VEL
LIN {X 0,Y 375.964,Z 512.649,A -85,B 0,C 180,E1 -12471.913,E2 -12471.913} C_VEL
LIN {X 0,Y 375.98,Z 512.643,A -85,B 0,C 180,E1 -12475.334,E2 -12475.334} C_VEL
LIN {X 0,Y 375.959,Z 512.648,A -85,B 0,C 180,E1 -12478.439,E2 -12478.439} C_VEL
LIN {X 0,Y 375.956,Z 512.683,A -85,B 0,C 180,E1 -12479.409,E2 -12479.409} C_VEL
LIN {X 0,Y 378.822,Z 524.87,A -85,B 0,C 180,E1 -12482.067,E2 -12482.067} C_VEL
LIN {X 0,Y 380.219,Z 532.512,A -85,B 0,C 180,E1 -12483.666,E2 -12483.666} C_VEL
LIN {X 0,Y 379.672,Z 544.818,A -85,B 0,C 180,E1 -12485.969,E2 -12485.969} C_VEL
LIN {X 0,Y 379.46,Z 548.664,A -85,B 0,C 180,E1 -12486.665,E2 -12486.665} C_VEL
LIN {X 0,Y 384.185,Z 573.266,A -85,B 0,C 180,E1 -12487.451,E2 -12487.451} C_VEL
LIN {X 0,Y 382.749,Z 659.032,A -85,B 0,C 180,E1 -12489.09,E2 -12489.09} C_VEL
LIN {X 0,Y 382.236,Z 672.277,A -85,B 0,C 180,E1 -12489.553,E2 -12489.553} C_VEL
LIN {X 0,Y 381.585,Z 685.725,A -85,B 0,C 180,E1 -12490.281,E2 -12490.281} C_VEL
LIN {X 0,Y 380.728,Z 697.676,A -85,B 0,C 180,E1 -12491.154,E2 -12491.154} C_VEL
LIN {X 0,Y 379.699,Z 708.904,A -85,B 0,C 180,E1 -12492.218,E2 -12492.218} C_VEL
LIN {X 0,Y 378.597,Z 719.054,A -85,B 0,C 180,E1 -12493.417,E2 -12493.417} C_VEL
LIN {X 0,Y 377.726,Z 727.372,A -85,B 0,C 180,E1 -12494.625,E2 -12494.625} C_VEL
LIN {X 0,Y 376.821,Z 736.378,A -85,B 0,C 180,E1 -12496.244,E2 -12496.244} C_VEL
LIN {X 0,Y 376.144,Z 743.599,A -85,B 0,C 180,E1 -12497.866,E2 -12497.866} C_VEL
LIN {X 0,Y 375.391,Z 750.227,A -85,B 0,C 180,E1 -12499.755,E2 -12499.755} C_VEL
LIN {X 0,Y 375.014,Z 754.568,A -85,B 0,C 180,E1 -12501.378,E2 -12501.378} C_VEL
LIN {X 0,Y 374.823,Z 756.85,A -85,B 0,C 180,E1 -12502.458,E2 -12502.458} C_VEL
LIN {X 0,Y 374.698,Z 759.054,A -85,B 0,C 180,E1 -12503.774,E2 -12503.774} C_VEL
LIN {X 0,Y 374.554,Z 761.119,A -85,B 0,C 180,E1 -12505.696,E2 -12505.696} C_VEL
LIN {X 0,Y 374.506,Z 761.959,A -85,B 0,C 180,E1 -12507.849,E2 -12507.849} C_VEL
LIN {X 0,Y 374.526,Z 761.759,A -85,B 0,C 180,E1 -12508.925,E2 -12508.925} C_VEL
LIN {X 0,Y 374.557,Z 761.168,A -85,B 0,C 180,E1 -12510,E2 -12510} C_VEL
LIN {X 0,Y 374.704,Z 758.825,A -85,B 0,C 180,E1 -12512.15,E2 -12512.15} C_VEL
LIN {X 0,Y 374.912,Z 755.948,A -85,B 0,C 180,E1 -12513.762,E2 -12513.762} C_VEL
LIN {X 0,Y 375.099,Z 752.047,A -85,B 0,C 180,E1 -12515.375,E2 -12515.375} C_VEL
LIN {X 0,Y 375.595,Z 746.739,A -85,B 0,C 180,E1 -12517.056,E2 -12517.056} C_VEL
LIN {X 0,Y 376.249,Z 739.438,A -85,B 0,C 180,E1 -12518.865,E2 -12518.865} C_VEL
LIN {X 0,Y 377.034,Z 731.246,A -85,B 0,C 180,E1 -12520.471,E2 -12520.471} C_VEL
LIN {X 0,Y 377.89,Z 722.81,A -85,B 0,C 180,E1 -12521.805,E2 -12521.805} C_VEL
LIN {X 0,Y 378.85,Z 712.133,A -85,B 0,C 180,E1 -12523.175,E2 -12523.175} C_VEL
LIN {X 0,Y 378.646,Z 707.444,A -85,B 0,C 180,E1 -12523.721,E2 -12523.721} C_VEL
LIN {X 0,Y 376.53,Z 699.634,A -85,B 0,C 180,E1 -12524.596,E2 -12524.596} C_VEL
LIN {X 0,Y 374.387,Z 691.415,A -85,B 0,C 180,E1 -12525.376,E2 -12525.376} C_VEL
LIN {X 0,Y 374.128,Z 686.09,A -85,B 0,C 180,E1 -12525.763,E2 -12525.763} C_VEL
LIN {X 0,Y 374.769,Z 672.949,A -85,B 0,C 180,E1 -12526.49,E2 -12526.49} C_VEL
LIN {X 0,Y 375.236,Z 660.514,A -85,B 0,C 180,E1 -12526.952,E2 -12526.952} C_VEL
LIN {X 0,Y 375.78,Z 629.76,A -85,B 0,C 180,E1 -12527.576,E2 -12527.576} C_VEL
LIN {X 0,Y 376.638,Z 573.936,A -85,B 0,C 180,E1 -12528.641,E2 -12528.641} C_VEL
LIN {X 0,Y 372.183,Z 548.804,A -85,B 0,C 180,E1 -12529.408,E2 -12529.408} C_VEL
LIN {X 0,Y 372.85,Z 534.074,A -85,B 0,C 180,E1 -12532.147,E2 -12532.147} C_VEL
LIN {X 0,Y 372.629,Z 530.949,A -85,B 0,C 180,E1 -12532.783,E2 -12532.783} C_VEL
LIN {X 0,Y 369.897,Z 517.513,A -85,B 0,C 180,E1 -12535.61,E2 -12535.61} C_VEL
LIN {X 0,Y 368.993,Z 513.525,A -85,B 0,C 180,E1 -12536.519,E2 -12536.519} C_VEL
LIN {X 0,Y 368.92,Z 513.534,A -85,B 0,C 180,E1 -12539.689,E2 -12539.689} C_VEL
LIN {X 0,Y 368.898,Z 513.534,A -85,B 0,C 180,E1 -12543.042,E2 -12543.042} C_VEL
LIN {X 0,Y 368.917,Z 513.528,A -85,B 0,C 180,E1 -12546.196,E2 -12546.196} C_VEL
LIN {X 0,Y 368.904,Z 513.533,A -85,B 0,C 180,E1 -12548.952,E2 -12548.952} C_VEL
LIN {X 0,Y 368.939,Z 513.526,A -85,B 0,C 180,E1 -12552.018,E2 -12552.018} C_VEL
LIN {X 0,Y 368.923,Z 513.519,A -85,B 0,C 180,E1 -12555.182,E2 -12555.182} C_VEL
LIN {X 0,Y 368.881,Z 513.534,A -85,B 0,C 180,E1 -12558.177,E2 -12558.177} C_VEL
LIN {X 0,Y 368.907,Z 513.533,A -85,B 0,C 180,E1 -12561.358,E2 -12561.358} C_VEL
LIN {X 0,Y 368.918,Z 513.613,A -85,B 0,C 180,E1 -12563.139,E2 -12563.139} C_VEL
LIN {X 0,Y 375.786,Z 532.772,A -85,B 0,C 180,E1 -12563.927,E2 -12563.927} C_VEL
LIN {X 0,Y 373.967,Z 617.388,A -85,B 0,C 180,E1 -12565.875,E2 -12565.875} C_VEL
LIN {X 0,Y 373.532,Z 631.312,A -85,B 0,C 180,E1 -12566.428,E2 -12566.428} C_VEL
LIN {X 0,Y 373.024,Z 643.406,A -85,B 0,C 180,E1 -12567.122,E2 -12567.122} C_VEL
LIN {X 0,Y 372.276,Z 656.076,A -85,B 0,C 180,E1 -12568.089,E2 -12568.089} C_VEL
LIN {X 0,Y 371.552,Z 666.828,A -85,B 0,C 180,E1 -12569.131,E2 -12569.131} C_VEL
LIN {X 0,Y 370.773,Z 677.84,A -85,B 0,C 180,E1 -12570.473,E2 -12570.473} C_VEL
LIN {X 0,Y 369.954,Z 687.66,A -85,B 0,C 180,E1 -12571.954,E2 -12571.954} C_VEL
LIN {X 0,Y 369.37,Z 695.488,A -85,B 0,C 180,E1 -12573.412,E2 -12573.412} C_VEL
LIN {X 0,Y 368.762,Z 703.22,A -85,B 0,C 180,E1 -12575.21,E2 -12575.21} C_VEL
LIN {X 0,Y 368.357,Z 709.193,A -85,B 0,C 180,E1 -12576.975,E2 -12576.975} C_VEL
LIN {X 0,Y 368.035,Z 713.724,A -85,B 0,C 180,E1 -12578.726,E2 -12578.726} C_VEL
LIN {X 0,Y 367.858,Z 716.012,A -85,B 0,C 180,E1 -12579.885,E2 -12579.885} C_VEL
LIN {X 0,Y 367.736,Z 717.823,A -85,B 0,C 180,E1 -12581.04,E2 -12581.04} C_VEL
LIN {X 0,Y 367.682,Z 719.7,A -85,B 0,C 180,E1 -12582.881,E2 -12582.881} C_VEL
LIN {X 0,Y 367.671,Z 720.356,A -85,B 0,C 180,E1 -12584.478,E2 -12584.478} C_VEL
LIN {X 0,Y 367.733,Z 720.281,A -85,B 0,C 180,E1 -12585.614,E2 -12585.614} C_VEL
LIN {X 0,Y 367.891,Z 719.601,A -85,B 0,C 180,E1 -12586.97,E2 -12586.97} C_VEL
LIN {X 0,Y 368.19,Z 717.397,A -85,B 0,C 180,E1 -12588.996,E2 -12588.996} C_VEL
LIN {X 0,Y 368.621,Z 714.407,A -85,B 0,C 180,E1 -12590.673,E2 -12590.673} C_VEL
LIN {X 0,Y 369.15,Z 710.316,A -85,B 0,C 180,E1 -12592.341,E2 -12592.341} C_VEL
LIN {X 0,Y 369.948,Z 704.01,A -85,B 0,C 180,E1 -12594.276,E2 -12594.276} C_VEL
LIN {X 0,Y 370.773,Z 697.118,A -85,B 0,C 180,E1 -12595.924,E2 -12595.924} C_VEL
LIN {X 0,Y 371.741,Z 688.504,A -85,B 0,C 180,E1 -12597.562,E2 -12597.562} C_VEL
LIN {X 0,Y 372.798,Z 679.64,A -85,B 0,C 180,E1 -12598.92,E2 -12598.92} C_VEL
LIN {X 0,Y 373.761,Z 669.966,A -85,B 0,C 180,E1 -12600.134,E2 -12600.134} C_VEL
LIN {X 0,Y 374.755,Z 659.273,A -85,B 0,C 180,E1 -12601.209,E2 -12601.209} C_VEL
LIN {X 0,Y 375.714,Z 647.455,A -85,B 0,C 180,E1 -12602.144,E2 -12602.144} C_VEL
LIN {X 0,Y 376.414,Z 635.419,A -85,B 0,C 180,E1 -12602.876,E2 -12602.876} C_VEL
LIN {X 0,Y 376.91,Z 622.307,A -85,B 0,C 180,E1 -12603.441,E2 -12603.441} C_VEL
LIN {X 0,Y 377.625,Z 597.16,A -85,B 0,C 180,E1 -12604.102,E2 -12604.102} C_VEL
LIN {X 0,Y 379.743,Z 537.749,A -85,B 0,C 180,E1 -12605.576,E2 -12605.576} C_VEL
LIN {X 0,Y 379.066,Z 535.696,A -85,B 0,C 180,E1 -12605.69,E2 -12605.69} C_VEL
LIN {X 0,Y 372.282,Z 520.837,A -85,B 0,C 180,E1 -12606.735,E2 -12606.735} C_VEL
LIN {X 0,Y 369.697,Z 515.658,A -85,B 0,C 180,E1 -12607.166,E2 -12607.166} C_VEL
LIN {X 0,Y 369.205,Z 513.497,A -85,B 0,C 180,E1 -12608.035,E2 -12608.035} C_VEL
LIN {X 0,Y 369.006,Z 513.52,A -85,B 0,C 180,E1 -12612.093,E2 -12612.093} C_VEL
LIN {X 0,Y 368.991,Z 513.524,A -85,B 0,C 180,E1 -12615.465,E2 -12615.465} C_VEL
LIN {X 0,Y 368.95,Z 513.528,A -85,B 0,C 180,E1 -12618.894,E2 -12618.894} C_VEL
LIN {X 0,Y 368.924,Z 513.529,A -85,B 0,C 180,E1 -12622.395,E2 -12622.395} C_VEL
LIN {X 0,Y 368.993,Z 513.518,A -85,B 0,C 180,E1 -12625.981,E2 -12625.981} C_VEL
LIN {X 0,Y 368.961,Z 513.524,A -85,B 0,C 180,E1 -12628.814,E2 -12628.814} C_VEL
LIN {X 0,Y 368.893,Z 513.528,A -85,B 0,C 180,E1 -12632.238,E2 -12632.238} C_VEL
LIN {X 0,Y 368.923,Z 513.531,A -85,B 0,C 180,E1 -12635.002,E2 -12635.002} C_VEL
LIN {X 0,Y 368.905,Z 513.531,A -85,B 0,C 180,E1 -12638.641,E2 -12638.641} C_VEL
LIN {X 0,Y 368.876,Z 513.534,A -85,B 0,C 180,E1 -12642.01,E2 -12642.01} C_VEL
LIN {X 0,Y 368.903,Z 513.535,A -85,B 0,C 180,E1 -12645.181,E2 -12645.181} C_VEL
LIN {X 0,Y 368.88,Z 513.539,A -85,B 0,C 180,E1 -12648.178,E2 -12648.178} C_VEL
LIN {X 0,Y 368.907,Z 513.534,A -85,B 0,C 180,E1 -12651.36,E2 -12651.36} C_VEL
LIN {X 0,Y 368.935,Z 513.532,A -85,B 0,C 180,E1 -12655.147,E2 -12655.147} C_VEL
LIN {X 0,Y 368.919,Z 513.568,A -85,B 0,C 180,E1 -12655.973,E2 -12655.973} C_VEL
LIN {X 0,Y 371.7,Z 524.01,A -85,B 0,C 180,E1 -12659.028,E2 -12659.028} C_VEL
LIN {X 0,Y 373.6,Z 532.701,A -85,B 0,C 180,E1 -12661.335,E2 -12661.335} C_VEL
LIN {X 0,Y 374.491,Z 537.901,A -85,B 0,C 180,E1 -12662.627,E2 -12662.627} C_VEL
LIN {X 0,Y 373.42,Z 547.796,A -85,B 0,C 180,E1 -12664.764,E2 -12664.764} C_VEL
LIN {X 0,Y 372.212,Z 559.082,A -85,B 0,C 180,E1 -12667.103,E2 -12667.103} C_VEL
LIN {X 0,Y 375.696,Z 577.99,A -85,B 0,C 180,E1 -12667.937,E2 -12667.937} C_VEL
LIN {X 0,Y 377.972,Z 597.56,A -85,B 0,C 180,E1 -12668.666,E2 -12668.666} C_VEL
LIN {X 0,Y 378.199,Z 603.473,A -85,B 0,C 180,E1 -12668.847,E2 -12668.847} C_VEL
LIN {X 0,Y 376.058,Z 671.529,A -85,B 0,C 180,E1 -12670.521,E2 -12670.521} C_VEL
LIN {X 0,Y 375.209,Z 685.46,A -85,B 0,C 180,E1 -12671.079,E2 -12671.079} C_VEL
LIN {X 0,Y 374.117,Z 698.055,A -85,B 0,C 180,E1 -12671.802,E2 -12671.802} C_VEL
LIN {X 0,Y 372.505,Z 715.562,A -85,B 0,C 180,E1 -12673.138,E2 -12673.138} C_VEL
LIN {X 0,Y 371.47,Z 727.335,A -85,B 0,C 180,E1 -12674.219,E2 -12674.219} C_VEL
LIN {X 0,Y 370.671,Z 737.515,A -85,B 0,C 180,E1 -12675.407,E2 -12675.407} C_VEL
LIN {X 0,Y 369.723,Z 747.298,A -85,B 0,C 180,E1 -12676.815,E2 -12676.815} C_VEL
LIN {X 0,Y 368.82,Z 756.37,A -85,B 0,C 180,E1 -12678.459,E2 -12678.459} C_VEL
LIN {X 0,Y 368.211,Z 763.66,A -85,B 0,C 180,E1 -12680.109,E2 -12680.109} C_VEL
LIN {X 0,Y 367.842,Z 769.478,A -85,B 0,C 180,E1 -12681.762,E2 -12681.762} C_VEL
LIN {X 0,Y 367.595,Z 774.031,A -85,B 0,C 180,E1 -12683.413,E2 -12683.413} C_VEL
LIN {X 0,Y 367.507,Z 776.418,A -85,B 0,C 180,E1 -12684.513,E2 -12684.513} C_VEL
LIN {X 0,Y 367.484,Z 778.371,A -85,B 0,C 180,E1 -12685.613,E2 -12685.613} C_VEL
LIN {X 0,Y 367.428,Z 779.898,A -85,B 0,C 180,E1 -12686.71,E2 -12686.71} C_VEL
LIN {X 0,Y 367.431,Z 780.965,A -85,B 0,C 180,E1 -12687.808,E2 -12687.808} C_VEL
LIN {X 0,Y 367.45,Z 781.632,A -85,B 0,C 180,E1 -12688.904,E2 -12688.904} C_VEL
LIN {X 0,Y 367.464,Z 781.908,A -85,B 0,C 180,E1 -12690,E2 -12690} C_VEL
LIN {X 0,Y 367.434,Z 781.777,A -85,B 0,C 180,E1 -12691.096,E2 -12691.096} C_VEL
LIN {X 0,Y 367.43,Z 781.208,A -85,B 0,C 180,E1 -12692.192,E2 -12692.192} C_VEL
LIN {X 0,Y 367.486,Z 778.891,A -85,B 0,C 180,E1 -12694.387,E2 -12694.387} C_VEL
LIN {X 0,Y 367.559,Z 775.824,A -85,B 0,C 180,E1 -12696.131,E2 -12696.131} C_VEL
LIN {X 0,Y 367.754,Z 772.089,A -85,B 0,C 180,E1 -12697.688,E2 -12697.688} C_VEL
LIN {X 0,Y 368.196,Z 766.017,A -85,B 0,C 180,E1 -12699.614,E2 -12699.614} C_VEL
LIN {X 0,Y 368.767,Z 759.358,A -85,B 0,C 180,E1 -12701.265,E2 -12701.265} C_VEL
LIN {X 0,Y 369.686,Z 751.093,A -85,B 0,C 180,E1 -12702.907,E2 -12702.907} C_VEL
LIN {X 0,Y 370.526,Z 742.56,A -85,B 0,C 180,E1 -12704.275,E2 -12704.275} C_VEL
LIN {X 0,Y 371.562,Z 732.021,A -85,B 0,C 180,E1 -12705.636,E2 -12705.636} C_VEL
LIN {X 0,Y 372.605,Z 721.552,A -85,B 0,C 180,E1 -12706.716,E2 -12706.716} C_VEL
LIN {X 0,Y 373.639,Z 709.884,A -85,B 0,C 180,E1 -12707.656,E2 -12707.656} C_VEL
LIN {X 0,Y 374.485,Z 697.749,A -85,B 0,C 180,E1 -12708.392,E2 -12708.392} C_VEL
LIN {X 0,Y 375.142,Z 685.364,A -85,B 0,C 180,E1 -12708.925,E2 -12708.925} C_VEL
LIN {X 0,Y 375.641,Z 672.668,A -85,B 0,C 180,E1 -12709.253,E2 -12709.253} C_VEL
LIN {X 0,Y 376.629,Z 600.185,A -85,B 0,C 180,E1 -12710.642,E2 -12710.642} C_VEL
LIN {X 0,Y 372.212,Z 567.283,A -85,B 0,C 180,E1 -12711.577,E2 -12711.577} C_VEL
LIN {X 0,Y 371.227,Z 560.203,A -85,B 0,C 180,E1 -12711.81,E2 -12711.81} C_VEL
LIN {X 0,Y 372.913,Z 540.602,A -85,B 0,C 180,E1 -12715.687,E2 -12715.687} C_VEL
LIN {X 0,Y 373.283,Z 534.769,A -85,B 0,C 180,E1 -12716.862,E2 -12716.862} C_VEL
LIN {X 0,Y 371.556,Z 525.648,A -85,B 0,C 180,E1 -12718.837,E2 -12718.837} C_VEL
LIN {X 0,Y 368.952,Z 513.529,A -85,B 0,C 180,E1 -12721.595,E2 -12721.595} C_VEL
LIN {X 0,Y 368.926,Z 513.532,A -85,B 0,C 180,E1 -12725.001,E2 -12725.001} C_VEL
LIN {X 0,Y 368.905,Z 513.503,A -85,B 0,C 180,E1 -12728.64,E2 -12728.64} C_VEL
LIN {X 0,Y 368.879,Z 513.535,A -85,B 0,C 180,E1 -12732.009,E2 -12732.009} C_VEL
LIN {X 0,Y 368.923,Z 513.531,A -85,B 0,C 180,E1 -12735.182,E2 -12735.182} C_VEL
LIN {X 0,Y 368.905,Z 513.522,A -85,B 0,C 180,E1 -12738.181,E2 -12738.181} C_VEL
LIN {X 0,Y 368.908,Z 513.532,A -85,B 0,C 180,E1 -12741.358,E2 -12741.358} C_VEL
LIN {X 0,Y 368.931,Z 513.527,A -85,B 0,C 180,E1 -12745.146,E2 -12745.146} C_VEL
LIN {X 0,Y 368.923,Z 513.517,A -85,B 0,C 180,E1 -12749.046,E2 -12749.046} C_VEL
LIN {X 0,Y 368.98,Z 513.523,A -85,B 0,C 180,E1 -12751.564,E2 -12751.564} C_VEL
LIN {X 0,Y 368.993,Z 513.515,A -85,B 0,C 180,E1 -12754.019,E2 -12754.019} C_VEL
LIN {X 0,Y 368.914,Z 513.525,A -85,B 0,C 180,E1 -12757.604,E2 -12757.604} C_VEL
LIN {X 0,Y 368.95,Z 513.522,A -85,B 0,C 180,E1 -12761.106,E2 -12761.106} C_VEL
LIN {X 0,Y 368.99,Z 513.505,A -85,B 0,C 180,E1 -12764.535,E2 -12764.535} C_VEL
LIN {X 0,Y 369.005,Z 513.517,A -85,B 0,C 180,E1 -12767.907,E2 -12767.907} C_VEL
LIN {X 0,Y 369.181,Z 513.476,A -85,B 0,C 180,E1 -12771.844,E2 -12771.844} C_VEL
LIN {X 0,Y 369.142,Z 513.498,A -85,B 0,C 180,E1 -12774.538,E2 -12774.538} C_VEL
LIN {X 0,Y 369.311,Z 513.473,A -85,B 0,C 180,E1 -12777.819,E2 -12777.819} C_VEL
LIN {X 0,Y 369.452,Z 513.438,A -85,B 0,C 180,E1 -12780,E2 -12780} C_VEL
LIN {X 0,Y 369.311,Z 513.473,A -85,B 0,C 180,E1 -12782.181,E2 -12782.181} C_VEL
LIN {X 0,Y 369.198,Z 513.49,A -85,B 0,C 180,E1 -12786.559,E2 -12786.559} C_VEL
LIN {X 0,Y 369.06,Z 513.503,A -85,B 0,C 180,E1 -12789.869,E2 -12789.869} C_VEL
LIN {X 0,Y 369.03,Z 513.511,A -85,B 0,C 180,E1 -12793.773,E2 -12793.773} C_VEL
LIN {X 0,Y 368.994,Z 513.514,A -85,B 0,C 180,E1 -12797.769,E2 -12797.769} C_VEL
LIN {X 0,Y 368.923,Z 513.526,A -85,B 0,C 180,E1 -12801.22,E2 -12801.22} C_VEL
LIN {X 0,Y 368.952,Z 513.518,A -85,B 0,C 180,E1 -12804.776,E2 -12804.776} C_VEL
LIN {X 0,Y 368.981,Z 513.518,A -85,B 0,C 180,E1 -12808.436,E2 -12808.436} C_VEL
LIN {X 0,Y 368.905,Z 513.531,A -85,B 0,C 180,E1 -12812.238,E2 -12812.238} C_VEL
LIN {X 0,Y 368.925,Z 513.523,A -85,B 0,C 180,E1 -12815.002,E2 -12815.002} C_VEL
LIN {X 0,Y 368.907,Z 513.533,A -85,B 0,C 180,E1 -12818.642,E2 -12818.642} C_VEL
LIN {X 0,Y 368.879,Z 513.538,A -85,B 0,C 180,E1 -12822.011,E2 -12822.011} C_VEL
LIN {X 0,Y 368.907,Z 513.537,A -85,B 0,C 180,E1 -12825.181,E2 -12825.181} C_VEL
LIN {X 0,Y 368.882,Z 513.534,A -85,B 0,C 180,E1 -12828.179,E2 -12828.179} C_VEL
LIN {X 0,Y 368.908,Z 513.531,A -85,B 0,C 180,E1 -12831.361,E2 -12831.361} C_VEL
LIN {X 0,Y 368.937,Z 513.52,A -85,B 0,C 180,E1 -12835.147,E2 -12835.147} C_VEL
LIN {X 0,Y 368.93,Z 513.68,A -85,B 0,C 180,E1 -12839.047,E2 -12839.047} C_VEL
LIN {X 0,Y 371.9,Z 526.166,A -85,B 0,C 180,E1 -12841.808,E2 -12841.808} C_VEL
LIN {X 0,Y 373.374,Z 533.898,A -85,B 0,C 180,E1 -12843.446,E2 -12843.446} C_VEL
LIN {X 0,Y 372.826,Z 546.341,A -85,B 0,C 180,E1 -12845.796,E2 -12845.796} C_VEL
LIN {X 0,Y 372.689,Z 548.834,A -85,B 0,C 180,E1 -12846.247,E2 -12846.247} C_VEL
LIN {X 0,Y 377.581,Z 574.129,A -85,B 0,C 180,E1 -12847.074,E2 -12847.074} C_VEL
LIN {X 0,Y 376.128,Z 658.295,A -85,B 0,C 180,E1 -12848.704,E2 -12848.704} C_VEL
LIN {X 0,Y 375.641,Z 671.146,A -85,B 0,C 180,E1 -12849.142,E2 -12849.142} C_VEL
LIN {X 0,Y 375.031,Z 683.098,A -85,B 0,C 180,E1 -12849.759,E2 -12849.759} C_VEL
LIN {X 0,Y 374.103,Z 695.917,A -85,B 0,C 180,E1 -12850.664,E2 -12850.664} C_VEL
LIN {X 0,Y 373.145,Z 706.314,A -85,B 0,C 180,E1 -12851.611,E2 -12851.611} C_VEL
LIN {X 0,Y 372.02,Z 716.988,A -85,B 0,C 180,E1 -12852.832,E2 -12852.832} C_VEL
LIN {X 0,Y 370.862,Z 727.414,A -85,B 0,C 180,E1 -12854.334,E2 -12854.334} C_VEL
LIN {X 0,Y 370.024,Z 735.106,A -85,B 0,C 180,E1 -12855.705,E2 -12855.705} C_VEL
LIN {X 0,Y 369.303,Z 742.606,A -85,B 0,C 180,E1 -12857.359,E2 -12857.359} C_VEL
LIN {X 0,Y 368.517,Z 748.619,A -85,B 0,C 180,E1 -12859.006,E2 -12859.006} C_VEL
LIN {X 0,Y 368.092,Z 753.368,A -85,B 0,C 180,E1 -12860.66,E2 -12860.66} C_VEL
LIN {X 0,Y 367.753,Z 756.998,A -85,B 0,C 180,E1 -12862.312,E2 -12862.312} C_VEL
LIN {X 0,Y 367.595,Z 759.433,A -85,B 0,C 180,E1 -12863.822,E2 -12863.822} C_VEL
LIN {X 0,Y 367.486,Z 761.294,A -85,B 0,C 180,E1 -12865.613,E2 -12865.613} C_VEL
LIN {X 0,Y 367.406,Z 762.148,A -85,B 0,C 180,E1 -12867.808,E2 -12867.808} C_VEL
LIN {X 0,Y 367.428,Z 761.96,A -85,B 0,C 180,E1 -12868.904,E2 -12868.904} C_VEL
LIN {X 0,Y 367.46,Z 761.375,A -85,B 0,C 180,E1 -12870,E2 -12870} C_VEL
LIN {X 0,Y 367.612,Z 759.049,A -85,B 0,C 180,E1 -12872.191,E2 -12872.191} C_VEL
LIN {X 0,Y 367.821,Z 756.185,A -85,B 0,C 180,E1 -12873.834,E2 -12873.834} C_VEL
LIN {X 0,Y 368.055,Z 752.297,A -85,B 0,C 180,E1 -12875.479,E2 -12875.479} C_VEL
LIN {X 0,Y 368.531,Z 747.414,A -85,B 0,C 180,E1 -12877.077,E2 -12877.077} C_VEL
LIN {X 0,Y 369.137,Z 740.921,A -85,B 0,C 180,E1 -12878.761,E2 -12878.761} C_VEL
LIN {X 0,Y 369.905,Z 733.031,A -85,B 0,C 180,E1 -12880.398,E2 -12880.398} C_VEL
LIN {X 0,Y 370.786,Z 724.967,A -85,B 0,C 180,E1 -12881.757,E2 -12881.757} C_VEL
LIN {X 0,Y 371.733,Z 715.096,A -85,B 0,C 180,E1 -12883.113,E2 -12883.113} C_VEL
LIN {X 0,Y 372.694,Z 704,A -85,B 0,C 180,E1 -12884.329,E2 -12884.329} C_VEL
LIN {X 0,Y 373.57,Z 693.148,A -85,B 0,C 180,E1 -12885.271,E2 -12885.271} C_VEL
LIN {X 0,Y 374.128,Z 686.09,A -85,B 0,C 180,E1 -12885.763,E2 -12885.763} C_VEL
LIN {X 0,Y 373.747,Z 682.475,A -85,B 0,C 180,E1 -12886.02,E2 -12886.02} C_VEL
LIN {X 0,Y 371.293,Z 676.876,A -85,B 0,C 180,E1 -12886.466,E2 -12886.466} C_VEL
LIN {X 0,Y 368.777,Z 671.187,A -85,B 0,C 180,E1 -12886.876,E2 -12886.876} C_VEL
LIN {X 0,Y 368.258,Z 667.432,A -85,B 0,C 180,E1 -12887.065,E2 -12887.065} C_VEL
LIN {X 0,Y 368.676,Z 653.602,A -85,B 0,C 180,E1 -12887.469,E2 -12887.469} C_VEL
LIN {X 0,Y 369.976,Z 574.949,A -85,B 0,C 180,E1 -12888.993,E2 -12888.993} C_VEL
LIN {X 0,Y 365.364,Z 548.846,A -85,B 0,C 180,E1 -12889.827,E2 -12889.827} C_VEL
LIN {X 0,Y 365.986,Z 534.159,A -85,B 0,C 180,E1 -12892.585,E2 -12892.585} C_VEL
LIN {X 0,Y 363.669,Z 522.06,A -85,B 0,C 180,E1 -12895.16,E2 -12895.16} C_VEL
LIN {X 0,Y 361.945,Z 514.402,A -85,B 0,C 180,E1 -12896.866,E2 -12896.866} C_VEL
LIN {X 0,Y 361.876,Z 514.412,A -85,B 0,C 180,E1 -12900.327,E2 -12900.327} C_VEL
LIN {X 0,Y 361.855,Z 514.408,A -85,B 0,C 180,E1 -12904.279,E2 -12904.279} C_VEL
LIN {X 0,Y 361.863,Z 514.407,A -85,B 0,C 180,E1 -12907.222,E2 -12907.222} C_VEL
LIN {X 0,Y 361.904,Z 514.397,A -85,B 0,C 180,E1 -12910.767,E2 -12910.767} C_VEL
LIN {X 0,Y 361.902,Z 514.398,A -85,B 0,C 180,E1 -12914.354,E2 -12914.354} C_VEL
LIN {X 0,Y 361.835,Z 514.412,A -85,B 0,C 180,E1 -12917.567,E2 -12917.567} C_VEL
LIN {X 0,Y 361.869,Z 514.409,A -85,B 0,C 180,E1 -12921.575,E2 -12921.575} C_VEL
LIN {X 0,Y 361.892,Z 514.409,A -85,B 0,C 180,E1 -12922.784,E2 -12922.784} C_VEL
LIN {X 0,Y 364.208,Z 521.302,A -85,B 0,C 180,E1 -12923.101,E2 -12923.101} C_VEL
LIN {X 0,Y 368.922,Z 534.183,A -85,B 0,C 180,E1 -12923.646,E2 -12923.646} C_VEL
LIN {X 0,Y 367.08,Z 617.716,A -85,B 0,C 180,E1 -12925.618,E2 -12925.618} C_VEL
LIN {X 0,Y 366.656,Z 631.168,A -85,B 0,C 180,E1 -12926.159,E2 -12926.159} C_VEL
LIN {X 0,Y 366.1,Z 644.114,A -85,B 0,C 180,E1 -12926.912,E2 -12926.912} C_VEL
LIN {X 0,Y 365.287,Z 657.008,A -85,B 0,C 180,E1 -12927.92,E2 -12927.92} C_VEL
LIN {X 0,Y 364.572,Z 667.453,A -85,B 0,C 180,E1 -12928.957,E2 -12928.957} C_VEL
LIN {X 0,Y 363.823,Z 677.677,A -85,B 0,C 180,E1 -12930.217,E2 -12930.217} C_VEL
LIN {X 0,Y 363.003,Z 687.35,A -85,B 0,C 180,E1 -12931.683,E2 -12931.683} C_VEL
LIN {X 0,Y 362.414,Z 695.138,A -85,B 0,C 180,E1 -12933.128,E2 -12933.128} C_VEL
LIN {X 0,Y 361.849,Z 702.107,A -85,B 0,C 180,E1 -12934.704,E2 -12934.704} C_VEL
LIN {X 0,Y 361.385,Z 708.618,A -85,B 0,C 180,E1 -12936.57,E2 -12936.57} C_VEL
LIN {X 0,Y 361.028,Z 713.274,A -85,B 0,C 180,E1 -12938.292,E2 -12938.292} C_VEL
LIN {X 0,Y 360.851,Z 715.817,A -85,B 0,C 180,E1 -12939.477,E2 -12939.477} C_VEL
LIN {X 0,Y 360.679,Z 717.778,A -85,B 0,C 180,E1 -12940.655,E2 -12940.655} C_VEL
LIN {X 0,Y 360.613,Z 720.095,A -85,B 0,C 180,E1 -12942.735,E2 -12942.735} C_VEL
LIN {X 0,Y 360.589,Z 720.828,A -85,B 0,C 180,E1 -12944.165,E2 -12944.165} C_VEL
LIN {X 0,Y 360.637,Z 720.93,A -85,B 0,C 180,E1 -12945.324,E2 -12945.324} C_VEL
LIN {X 0,Y 360.829,Z 720.344,A -85,B 0,C 180,E1 -12946.867,E2 -12946.867} C_VEL
LIN {X 0,Y 361.086,Z 718.523,A -85,B 0,C 180,E1 -12948.776,E2 -12948.776} C_VEL
LIN {X 0,Y 361.53,Z 715.78,A -85,B 0,C 180,E1 -12950.489,E2 -12950.489} C_VEL
LIN {X 0,Y 362.063,Z 711.971,A -85,B 0,C 180,E1 -12952.19,E2 -12952.19} C_VEL
LIN {X 0,Y 362.736,Z 707.008,A -85,B 0,C 180,E1 -12953.883,E2 -12953.883} C_VEL
LIN {X 0,Y 363.568,Z 700.711,A -85,B 0,C 180,E1 -12955.565,E2 -12955.565} C_VEL
LIN {X 0,Y 364.51,Z 692.837,A -85,B 0,C 180,E1 -12957.237,E2 -12957.237} C_VEL
LIN {X 0,Y 365.557,Z 684.922,A -85,B 0,C 180,E1 -12958.595,E2 -12958.595} C_VEL
LIN {X 0,Y 366.65,Z 674.951,A -85,B 0,C 180,E1 -12960,E2 -12960} C_VEL
LIN {X 0,Y 367.846,Z 663.874,A -85,B 0,C 180,E1 -12961.231,E2 -12961.231} C_VEL
LIN {X 0,Y 368.812,Z 653.236,A -85,B 0,C 180,E1 -12962.184,E2 -12962.184} C_VEL
LIN {X 0,Y 369.695,Z 640.591,A -85,B 0,C 180,E1 -12963.065,E2 -12963.065} C_VEL
LIN {X 0,Y 370.358,Z 627.135,A -85,B 0,C 180,E1 -12963.74,E2 -12963.74} C_VEL
LIN {X 0,Y 370.784,Z 613.72,A -85,B 0,C 180,E1 -12964.178,E2 -12964.178} C_VEL
LIN {X 0,Y 373.433,Z 539.152,A -85,B 0,C 180,E1 -12966.077,E2 -12966.077} C_VEL
LIN {X 0,Y 366.775,Z 524.406,A -85,B 0,C 180,E1 -12967.153,E2 -12967.153} C_VEL
LIN {X 0,Y 362.662,Z 516.527,A -85,B 0,C 180,E1 -12967.857,E2 -12967.857} C_VEL
LIN {X 0,Y 362.099,Z 514.382,A -85,B 0,C 180,E1 -12968.807,E2 -12968.807} C_VEL
LIN {X 0,Y 361.959,Z 514.398,A -85,B 0,C 180,E1 -12972.332,E2 -12972.332} C_VEL
LIN {X 0,Y 361.955,Z 514.4,A -85,B 0,C 180,E1 -12974.62,E2 -12974.62} C_VEL
LIN {X 0,Y 361.948,Z 514.397,A -85,B 0,C 180,E1 -12978.1,E2 -12978.1} C_VEL
LIN {X 0,Y 361.884,Z 514.405,A -85,B 0,C 180,E1 -12981.653,E2 -12981.653} C_VEL
LIN {X 0,Y 361.921,Z 514.4,A -85,B 0,C 180,E1 -12985.29,E2 -12985.29} C_VEL
LIN {X 0,Y 361.916,Z 514.397,A -85,B 0,C 180,E1 -12987.778,E2 -12987.778} C_VEL
LIN {X 0,Y 361.84,Z 514.408,A -85,B 0,C 180,E1 -12991.286,E2 -12991.286} C_VEL
LIN {X 0,Y 361.848,Z 514.406,A -85,B 0,C 180,E1 -12994.281,E2 -12994.281} C_VEL
LIN {X 0,Y 361.859,Z 514.411,A -85,B 0,C 180,E1 -12997.224,E2 -12997.224} C_VEL
LIN {X 0,Y 361.831,Z 514.413,A -85,B 0,C 180,E1 -13000.756,E2 -13000.756} C_VEL
LIN {X 0,Y 361.829,Z 514.413,A -85,B 0,C 180,E1 -13004.367,E2 -13004.367} C_VEL
LIN {X 0,Y 361.833,Z 514.415,A -85,B 0,C 180,E1 -13007.569,E2 -13007.569} C_VEL
LIN {X 0,Y 361.868,Z 514.413,A -85,B 0,C 180,E1 -13010.974,E2 -13010.974} C_VEL
LIN {X 0,Y 361.872,Z 514.412,A -85,B 0,C 180,E1 -13014.656,E2 -13014.656} C_VEL
LIN {X 0,Y 361.924,Z 514.529,A -85,B 0,C 180,E1 -13015.264,E2 -13015.264} C_VEL
LIN {X 0,Y 364.324,Z 523.61,A -85,B 0,C 180,E1 -13018.08,E2 -13018.08} C_VEL
LIN {X 0,Y 366.324,Z 531.816,A -85,B 0,C 180,E1 -13020.396,E2 -13020.396} C_VEL
LIN {X 0,Y 367.714,Z 539.745,A -85,B 0,C 180,E1 -13022.449,E2 -13022.449} C_VEL
LIN {X 0,Y 366.571,Z 549.58,A -85,B 0,C 180,E1 -13024.631,E2 -13024.631} C_VEL
LIN {X 0,Y 365.588,Z 558.086,A -85,B 0,C 180,E1 -13026.459,E2 -13026.459} C_VEL
LIN {X 0,Y 369.305,Z 578.126,A -85,B 0,C 180,E1 -13027.409,E2 -13027.409} C_VEL
LIN {X 0,Y 371.506,Z 596.919,A -85,B 0,C 180,E1 -13028.137,E2 -13028.137} C_VEL
LIN {X 0,Y 371.869,Z 603.751,A -85,B 0,C 180,E1 -13028.361,E2 -13028.361} C_VEL
LIN {X 0,Y 369.581,Z 670.644,A -85,B 0,C 180,E1 -13030.057,E2 -13030.057} C_VEL
LIN {X 0,Y 368.747,Z 683.783,A -85,B 0,C 180,E1 -13030.589,E2 -13030.589} C_VEL
LIN {X 0,Y 367.616,Z 696.683,A -85,B 0,C 180,E1 -13031.324,E2 -13031.324} C_VEL
LIN {X 0,Y 366.355,Z 709.096,A -85,B 0,C 180,E1 -13032.27,E2 -13032.27} C_VEL
LIN {X 0,Y 364.759,Z 725.721,A -85,B 0,C 180,E1 -13033.777,E2 -13033.777} C_VEL
LIN {X 0,Y 363.822,Z 736.157,A -85,B 0,C 180,E1 -13034.985,E2 -13034.985} C_VEL
LIN {X 0,Y 362.943,Z 745.245,A -85,B 0,C 180,E1 -13036.279,E2 -13036.279} C_VEL
LIN {X 0,Y 362.143,Z 753.3,A -85,B 0,C 180,E1 -13037.674,E2 -13037.674} C_VEL
LIN {X 0,Y 361.421,Z 761.173,A -85,B 0,C 180,E1 -13039.355,E2 -13039.355} C_VEL
LIN {X 0,Y 360.904,Z 767.429,A -85,B 0,C 180,E1 -13041.038,E2 -13041.038} C_VEL
LIN {X 0,Y 360.6,Z 772.389,A -85,B 0,C 180,E1 -13042.722,E2 -13042.722} C_VEL
LIN {X 0,Y 360.428,Z 776.198,A -85,B 0,C 180,E1 -13044.405,E2 -13044.405} C_VEL
LIN {X 0,Y 360.393,Z 778.155,A -85,B 0,C 180,E1 -13045.526,E2 -13045.526} C_VEL
LIN {X 0,Y 360.345,Z 779.689,A -85,B 0,C 180,E1 -13046.646,E2 -13046.646} C_VEL
LIN {X 0,Y 360.331,Z 780.763,A -85,B 0,C 180,E1 -13047.764,E2 -13047.764} C_VEL
LIN {X 0,Y 360.351,Z 781.434,A -85,B 0,C 180,E1 -13048.883,E2 -13048.883} C_VEL
LIN {X 0,Y 360.367,Z 781.715,A -85,B 0,C 180,E1 -13050,E2 -13050} C_VEL
LIN {X 0,Y 360.335,Z 781.591,A -85,B 0,C 180,E1 -13051.118,E2 -13051.118} C_VEL
LIN {X 0,Y 360.331,Z 781.029,A -85,B 0,C 180,E1 -13052.236,E2 -13052.236} C_VEL
LIN {X 0,Y 360.346,Z 780.073,A -85,B 0,C 180,E1 -13053.354,E2 -13053.354} C_VEL
LIN {X 0,Y 360.395,Z 778.721,A -85,B 0,C 180,E1 -13054.474,E2 -13054.474} C_VEL
LIN {X 0,Y 360.464,Z 775.972,A -85,B 0,C 180,E1 -13056.091,E2 -13056.091} C_VEL
LIN {X 0,Y 360.696,Z 771.938,A -85,B 0,C 180,E1 -13057.839,E2 -13057.839} C_VEL
LIN {X 0,Y 361.065,Z 766.874,A -85,B 0,C 180,E1 -13059.523,E2 -13059.523} C_VEL
LIN {X 0,Y 361.641,Z 760.468,A -85,B 0,C 180,E1 -13061.206,E2 -13061.206} C_VEL
LIN {X 0,Y 362.565,Z 752.472,A -85,B 0,C 180,E1 -13062.88,E2 -13062.88} C_VEL
LIN {X 0,Y 363.437,Z 744.304,A -85,B 0,C 180,E1 -13064.273,E2 -13064.273} C_VEL
LIN {X 0,Y 364.517,Z 734.302,A -85,B 0,C 180,E1 -13065.659,E2 -13065.659} C_VEL
LIN {X 0,Y 365.528,Z 724.363,A -85,B 0,C 180,E1 -13066.762,E2 -13066.762} C_VEL
LIN {X 0,Y 366.542,Z 713.542,A -85,B 0,C 180,E1 -13067.721,E2 -13067.721} C_VEL
LIN {X 0,Y 367.505,Z 701.581,A -85,B 0,C 180,E1 -13068.537,E2 -13068.537} C_VEL
LIN {X 0,Y 368.306,Z 689.21,A -85,B 0,C 180,E1 -13069.145,E2 -13069.145} C_VEL
LIN {X 0,Y 368.862,Z 676.371,A -85,B 0,C 180,E1 -13069.549,E2 -13069.549} C_VEL
LIN {X 0,Y 370.008,Z 600.703,A -85,B 0,C 180,E1 -13071.033,E2 -13071.033} C_VEL
LIN {X 0,Y 365.806,Z 569.138,A -85,B 0,C 180,E1 -13071.951,E2 -13071.951} C_VEL
LIN {X 0,Y 364.461,Z 560.265,A -85,B 0,C 180,E1 -13072.241,E2 -13072.241} C_VEL
LIN {X 0,Y 364.376,Z 558.679,A -85,B 0,C 180,E1 -13072.361,E2 -13072.361} C_VEL
LIN {X 0,Y 366.13,Z 539.68,A -85,B 0,C 180,E1 -13076.199,E2 -13076.199} C_VEL
LIN {X 0,Y 366.227,Z 535.274,A -85,B 0,C 180,E1 -13077.114,E2 -13077.114} C_VEL
LIN {X 0,Y 363.765,Z 523.143,A -85,B 0,C 180,E1 -13079.823,E2 -13079.823} C_VEL
LIN {X 0,Y 361.891,Z 514.408,A -85,B 0,C 180,E1 -13081.869,E2 -13081.869} C_VEL
LIN {X 0,Y 361.865,Z 514.406,A -85,B 0,C 180,E1 -13085.636,E2 -13085.636} C_VEL
LIN {X 0,Y 361.866,Z 514.382,A -85,B 0,C 180,E1 -13089.026,E2 -13089.026} C_VEL
LIN {X 0,Y 361.833,Z 514.412,A -85,B 0,C 180,E1 -13092.828,E2 -13092.828} C_VEL
LIN {X 0,Y 361.853,Z 514.411,A -85,B 0,C 180,E1 -13095.939,E2 -13095.939} C_VEL
LIN {X 0,Y 361.867,Z 514.404,A -85,B 0,C 180,E1 -13099.237,E2 -13099.237} C_VEL
LIN {X 0,Y 361.868,Z 514.4,A -85,B 0,C 180,E1 -13102.982,E2 -13102.982} C_VEL
LIN {X 0,Y 361.853,Z 514.411,A -85,B 0,C 180,E1 -13106.63,E2 -13106.63} C_VEL
LIN {X 0,Y 361.87,Z 514.396,A -85,B 0,C 180,E1 -13109.672,E2 -13109.672} C_VEL
LIN {X 0,Y 361.948,Z 514.395,A -85,B 0,C 180,E1 -13113.475,E2 -13113.475} C_VEL
LIN {X 0,Y 361.872,Z 514.394,A -85,B 0,C 180,E1 -13117.144,E2 -13117.144} C_VEL
LIN {X 0,Y 361.899,Z 514.404,A -85,B 0,C 180,E1 -13120.723,E2 -13120.723} C_VEL
LIN {X 0,Y 361.924,Z 514.382,A -85,B 0,C 180,E1 -13123.066,E2 -13123.066} C_VEL
LIN {X 0,Y 361.992,Z 514.39,A -85,B 0,C 180,E1 -13126.528,E2 -13126.528} C_VEL
LIN {X 0,Y 362.028,Z 514.377,A -85,B 0,C 180,E1 -13129.938,E2 -13129.938} C_VEL
LIN {X 0,Y 362.161,Z 514.36,A -85,B 0,C 180,E1 -13133.314,E2 -13133.314} C_VEL
LIN {X 0,Y 362.275,Z 514.35,A -85,B 0,C 180,E1 -13137.777,E2 -13137.777} C_VEL
LIN {X 0,Y 362.421,Z 514.313,A -85,B 0,C 180,E1 -13140,E2 -13140} C_VEL
LIN {X 0,Y 362.276,Z 514.349,A -85,B 0,C 180,E1 -13142.224,E2 -13142.224} C_VEL
LIN {X 0,Y 362.159,Z 514.363,A -85,B 0,C 180,E1 -13146.687,E2 -13146.687} C_VEL
LIN {X 0,Y 362.024,Z 514.379,A -85,B 0,C 180,E1 -13150.063,E2 -13150.063} C_VEL
LIN {X 0,Y 361.991,Z 514.388,A -85,B 0,C 180,E1 -13153.899,E2 -13153.899} C_VEL
LIN {X 0,Y 361.961,Z 514.39,A -85,B 0,C 180,E1 -13157.939,E2 -13157.939} C_VEL
LIN {X 0,Y 361.886,Z 514.399,A -85,B 0,C 180,E1 -13161.654,E2 -13161.654} C_VEL
LIN {X 0,Y 361.922,Z 514.4,A -85,B 0,C 180,E1 -13165.291,E2 -13165.291} C_VEL
LIN {X 0,Y 361.917,Z 514.398,A -85,B 0,C 180,E1 -13167.779,E2 -13167.779} C_VEL
LIN {X 0,Y 361.855,Z 514.41,A -85,B 0,C 180,E1 -13171.628,E2 -13171.628} C_VEL
LIN {X 0,Y 361.871,Z 514.402,A -85,B 0,C 180,E1 -13175.346,E2 -13175.346} C_VEL
LIN {X 0,Y 361.867,Z 514.406,A -85,B 0,C 180,E1 -13179.028,E2 -13179.028} C_VEL
LIN {X 0,Y 361.834,Z 514.414,A -85,B 0,C 180,E1 -13182.83,E2 -13182.83} C_VEL
LIN {X 0,Y 361.828,Z 514.414,A -85,B 0,C 180,E1 -13185.946,E2 -13185.946} C_VEL
LIN {X 0,Y 361.835,Z 514.411,A -85,B 0,C 180,E1 -13189.246,E2 -13189.246} C_VEL
LIN {X 0,Y 361.864,Z 514.41,A -85,B 0,C 180,E1 -13192.778,E2 -13192.778} C_VEL
LIN {X 0,Y 361.855,Z 514.405,A -85,B 0,C 180,E1 -13195.721,E2 -13195.721} C_VEL
LIN {X 0,Y 361.931,Z 514.59,A -85,B 0,C 180,E1 -13198.655,E2 -13198.655} C_VEL
LIN {X 0,Y 364.98,Z 527.296,A -85,B 0,C 180,E1 -13201.504,E2 -13201.504} C_VEL
LIN {X 0,Y 366.52,Z 535.315,A -85,B 0,C 180,E1 -13203.218,E2 -13203.218} C_VEL
LIN {X 0,Y 366.24,Z 543.484,A -85,B 0,C 180,E1 -13204.796,E2 -13204.796} C_VEL
LIN {X 0,Y 365.931,Z 548.952,A -85,B 0,C 180,E1 -13205.802,E2 -13205.802} C_VEL
LIN {X 0,Y 370.936,Z 574.832,A -85,B 0,C 180,E1 -13206.677,E2 -13206.677} C_VEL
LIN {X 0,Y 369.468,Z 658.862,A -85,B 0,C 180,E1 -13208.338,E2 -13208.338} C_VEL
LIN {X 0,Y 368.96,Z 671.586,A -85,B 0,C 180,E1 -13208.783,E2 -13208.783} C_VEL
LIN {X 0,Y 368.245,Z 684.62,A -85,B 0,C 180,E1 -13209.485,E2 -13209.485} C_VEL
LIN {X 0,Y 367.377,Z 695.815,A -85,B 0,C 180,E1 -13210.296,E2 -13210.296} C_VEL
LIN {X 0,Y 366.399,Z 706.268,A -85,B 0,C 180,E1 -13211.26,E2 -13211.26} C_VEL
LIN {X 0,Y 365.234,Z 717.001,A -85,B 0,C 180,E1 -13212.503,E2 -13212.503} C_VEL
LIN {X 0,Y 364.003,Z 727.458,A -85,B 0,C 180,E1 -13214.03,E2 -13214.03} C_VEL
LIN {X 0,Y 362.97,Z 736.397,A -85,B 0,C 180,E1 -13215.678,E2 -13215.678} C_VEL
LIN {X 0,Y 362.23,Z 743.797,A -85,B 0,C 180,E1 -13217.393,E2 -13217.393} C_VEL
LIN {X 0,Y 361.359,Z 750.477,A -85,B 0,C 180,E1 -13219.353,E2 -13219.353} C_VEL
LIN {X 0,Y 360.945,Z 754.849,A -85,B 0,C 180,E1 -13221.039,E2 -13221.039} C_VEL
LIN {X 0,Y 360.695,Z 757.146,A -85,B 0,C 180,E1 -13222.161,E2 -13222.161} C_VEL
LIN {X 0,Y 360.513,Z 759.771,A -85,B 0,C 180,E1 -13223.84,E2 -13223.84} C_VEL
LIN {X 0,Y 360.397,Z 761.469,A -85,B 0,C 180,E1 -13225.526,E2 -13225.526} C_VEL
LIN {X 0,Y 360.307,Z 762.337,A -85,B 0,C 180,E1 -13227.764,E2 -13227.764} C_VEL
LIN {X 0,Y 360.329,Z 762.16,A -85,B 0,C 180,E1 -13228.882,E2 -13228.882} C_VEL
LIN {X 0,Y 360.362,Z 761.582,A -85,B 0,C 180,E1 -13230,E2 -13230} C_VEL
LIN {X 0,Y 360.519,Z 759.273,A -85,B 0,C 180,E1 -13232.234,E2 -13232.234} C_VEL
LIN {X 0,Y 360.732,Z 756.42,A -85,B 0,C 180,E1 -13233.91,E2 -13233.91} C_VEL
LIN {X 0,Y 361.014,Z 752.546,A -85,B 0,C 180,E1 -13235.586,E2 -13235.586} C_VEL
LIN {X 0,Y 361.588,Z 746.424,A -85,B 0,C 180,E1 -13237.575,E2 -13237.575} C_VEL
LIN {X 0,Y 362.23,Z 740.009,A -85,B 0,C 180,E1 -13239.211,E2 -13239.211} C_VEL
LIN {X 0,Y 363.107,Z 731.873,A -85,B 0,C 180,E1 -13240.877,E2 -13240.877} C_VEL
LIN {X 0,Y 364.032,Z 723.484,A -85,B 0,C 180,E1 -13242.261,E2 -13242.261} C_VEL
LIN {X 0,Y 365.045,Z 713.199,A -85,B 0,C 180,E1 -13243.641,E2 -13243.641} C_VEL
LIN {X 0,Y 366.015,Z 703.027,A -85,B 0,C 180,E1 -13244.739,E2 -13244.739} C_VEL
LIN {X 0,Y 366.908,Z 691.807,A -85,B 0,C 180,E1 -13245.697,E2 -13245.697} C_VEL
LIN {X 0,Y 367.804,Z 679.14,A -85,B 0,C 180,E1 -13246.513,E2 -13246.513} C_VEL
LIN {X 0,Y 368.258,Z 667.432,A -85,B 0,C 180,E1 -13247.065,E2 -13247.065} C_VEL
LIN {X 0,Y 367.867,Z 661.737,A -85,B 0,C 180,E1 -13247.3,E2 -13247.3} C_VEL
LIN {X 0,Y 363.254,Z 644.98,A -85,B 0,C 180,E1 -13247.946,E2 -13247.946} C_VEL
LIN {X 0,Y 362.377,Z 639.214,A -85,B 0,C 180,E1 -13248.105,E2 -13248.105} C_VEL
LIN {X 0,Y 362.338,Z 637.26,A -85,B 0,C 180,E1 -13248.146,E2 -13248.146} C_VEL
LIN {X 0,Y 363.331,Z 575.921,A -85,B 0,C 180,E1 -13249.359,E2 -13249.359} C_VEL
LIN {X 0,Y 358.65,Z 549.658,A -85,B 0,C 180,E1 -13250.194,E2 -13250.194} C_VEL
LIN {X 0,Y 358.59,Z 548.675,A -85,B 0,C 180,E1 -13250.296,E2 -13250.296} C_VEL
LIN {X 0,Y 359.107,Z 535.488,A -85,B 0,C 180,E1 -13252.8,E2 -13252.8} C_VEL
LIN {X 0,Y 356.898,Z 524.022,A -85,B 0,C 180,E1 -13255.281,E2 -13255.281} C_VEL
LIN {X 0,Y 354.903,Z 515.277,A -85,B 0,C 180,E1 -13257.253,E2 -13257.253} C_VEL
LIN {X 0,Y 354.855,Z 515.286,A -85,B 0,C 180,E1 -13259.678,E2 -13259.678} C_VEL
LIN {X 0,Y 354.807,Z 515.285,A -85,B 0,C 180,E1 -13263.701,E2 -13263.701} C_VEL
LIN {X 0,Y 354.797,Z 515.285,A -85,B 0,C 180,E1 -13266.458,E2 -13266.458} C_VEL
LIN {X 0,Y 354.823,Z 515.282,A -85,B 0,C 180,E1 -13269.423,E2 -13269.423} C_VEL
LIN {X 0,Y 354.832,Z 515.288,A -85,B 0,C 180,E1 -13272.874,E2 -13272.874} C_VEL
LIN {X 0,Y 354.782,Z 515.282,A -85,B 0,C 180,E1 -13276.105,E2 -13276.105} C_VEL
LIN {X 0,Y 354.786,Z 515.293,A -85,B 0,C 180,E1 -13279.178,E2 -13279.178} C_VEL
LIN {X 0,Y 354.823,Z 515.289,A -85,B 0,C 180,E1 -13282.485,E2 -13282.485} C_VEL
LIN {X 0,Y 362.146,Z 535.779,A -85,B 0,C 180,E1 -13283.37,E2 -13283.37} C_VEL
LIN {X 0,Y 360.149,Z 618.42,A -85,B 0,C 180,E1 -13285.379,E2 -13285.379} C_VEL
LIN {X 0,Y 359.752,Z 631.443,A -85,B 0,C 180,E1 -13285.914,E2 -13285.914} C_VEL
LIN {X 0,Y 359.151,Z 644.604,A -85,B 0,C 180,E1 -13286.692,E2 -13286.692} C_VEL
LIN {X 0,Y 358.334,Z 657.557,A -85,B 0,C 180,E1 -13287.724,E2 -13287.724} C_VEL
LIN {X 0,Y 357.596,Z 667.972,A -85,B 0,C 180,E1 -13288.777,E2 -13288.777} C_VEL
LIN {X 0,Y 356.757,Z 679.025,A -85,B 0,C 180,E1 -13290.178,E2 -13290.178} C_VEL
LIN {X 0,Y 355.922,Z 688.812,A -85,B 0,C 180,E1 -13291.712,E2 -13291.712} C_VEL
LIN {X 0,Y 355.243,Z 696.755,A -85,B 0,C 180,E1 -13293.251,E2 -13293.251} C_VEL
LIN {X 0,Y 354.653,Z 704.378,A -85,B 0,C 180,E1 -13295.095,E2 -13295.095} C_VEL
LIN {X 0,Y 354.288,Z 709.447,A -85,B 0,C 180,E1 -13296.625,E2 -13296.625} C_VEL
LIN {X 0,Y 353.916,Z 714.208,A -85,B 0,C 180,E1 -13298.447,E2 -13298.447} C_VEL
LIN {X 0,Y 353.646,Z 717.691,A -85,B 0,C 180,E1 -13300.254,E2 -13300.254} C_VEL
LIN {X 0,Y 353.555,Z 719.356,A -85,B 0,C 180,E1 -13301.455,E2 -13301.455} C_VEL
LIN {X 0,Y 353.548,Z 720.536,A -85,B 0,C 180,E1 -13302.651,E2 -13302.651} C_VEL
LIN {X 0,Y 353.531,Z 721.28,A -85,B 0,C 180,E1 -13303.84,E2 -13303.84} C_VEL
LIN {X 0,Y 353.554,Z 721.528,A -85,B 0,C 180,E1 -13305.024,E2 -13305.024} C_VEL
LIN {X 0,Y 353.76,Z 721.086,A -85,B 0,C 180,E1 -13306.765,E2 -13306.765} C_VEL
LIN {X 0,Y 353.984,Z 719.623,A -85,B 0,C 180,E1 -13308.548,E2 -13308.548} C_VEL
LIN {X 0,Y 354.272,Z 718.076,A -85,B 0,C 180,E1 -13309.715,E2 -13309.715} C_VEL
LIN {X 0,Y 354.803,Z 714.894,A -85,B 0,C 180,E1 -13311.457,E2 -13311.457} C_VEL
LIN {X 0,Y 355.42,Z 710.612,A -85,B 0,C 180,E1 -13313.186,E2 -13313.186} C_VEL
LIN {X 0,Y 356.181,Z 705.111,A -85,B 0,C 180,E1 -13314.906,E2 -13314.906} C_VEL
LIN {X 0,Y 357.175,Z 698.166,A -85,B 0,C 180,E1 -13316.616,E2 -13316.616} C_VEL
LIN {X 0,Y 358.31,Z 689.487,A -85,B 0,C 180,E1 -13318.314,E2 -13318.314} C_VEL
LIN {X 0,Y 359.55,Z 680.378,A -85,B 0,C 180,E1 -13319.752,E2 -13319.752} C_VEL
LIN {X 0,Y 360.622,Z 670.877,A -85,B 0,C 180,E1 -13320.977,E2 -13320.977} C_VEL
LIN {X 0,Y 361.872,Z 658.653,A -85,B 0,C 180,E1 -13322.226,E2 -13322.226} C_VEL
LIN {X 0,Y 362.959,Z 646.357,A -85,B 0,C 180,E1 -13323.191,E2 -13323.191} C_VEL
LIN {X 0,Y 363.735,Z 632.888,A -85,B 0,C 180,E1 -13323.981,E2 -13323.981} C_VEL
LIN {X 0,Y 364.309,Z 620.005,A -85,B 0,C 180,E1 -13324.495,E2 -13324.495} C_VEL
LIN {X 0,Y 367.335,Z 541.503,A -85,B 0,C 180,E1 -13326.57,E2 -13326.57} C_VEL
LIN {X 0,Y 361.134,Z 527.606,A -85,B 0,C 180,E1 -13327.622,E2 -13327.622} C_VEL
LIN {X 0,Y 355.63,Z 517.447,A -85,B 0,C 180,E1 -13328.578,E2 -13328.578} C_VEL
LIN {X 0,Y 355,Z 515.267,A -85,B 0,C 180,E1 -13329.544,E2 -13329.544} C_VEL
LIN {X 0,Y 354.944,Z 515.272,A -85,B 0,C 180,E1 -13333.745,E2 -13333.745} C_VEL
LIN {X 0,Y 354.891,Z 515.281,A -85,B 0,C 180,E1 -13337.28,E2 -13337.28} C_VEL
LIN {X 0,Y 354.832,Z 515.288,A -85,B 0,C 180,E1 -13340.886,E2 -13340.886} C_VEL
LIN {X 0,Y 354.854,Z 515.282,A -85,B 0,C 180,E1 -13344.577,E2 -13344.577} C_VEL
LIN {X 0,Y 354.878,Z 515.277,A -85,B 0,C 180,E1 -13347.096,E2 -13347.096} C_VEL
LIN {X 0,Y 354.848,Z 515.277,A -85,B 0,C 180,E1 -13349.679,E2 -13349.679} C_VEL
LIN {X 0,Y 354.8,Z 515.284,A -85,B 0,C 180,E1 -13353.703,E2 -13353.703} C_VEL
LIN {X 0,Y 354.793,Z 515.286,A -85,B 0,C 180,E1 -13356.46,E2 -13356.46} C_VEL
LIN {X 0,Y 354.819,Z 515.287,A -85,B 0,C 180,E1 -13359.424,E2 -13359.424} C_VEL
LIN {X 0,Y 354.784,Z 515.293,A -85,B 0,C 180,E1 -13362.868,E2 -13362.868} C_VEL
LIN {X 0,Y 354.772,Z 515.294,A -85,B 0,C 180,E1 -13366.106,E2 -13366.106} C_VEL
LIN {X 0,Y 354.785,Z 515.294,A -85,B 0,C 180,E1 -13369.18,E2 -13369.18} C_VEL
LIN {X 0,Y 354.809,Z 515.291,A -85,B 0,C 180,E1 -13372.402,E2 -13372.402} C_VEL
LIN {X 0,Y 354.845,Z 515.363,A -85,B 0,C 180,E1 -13374.448,E2 -13374.448} C_VEL
LIN {X 0,Y 357.562,Z 525.264,A -85,B 0,C 180,E1 -13377.691,E2 -13377.691} C_VEL
LIN {X 0,Y 359.782,Z 534.809,A -85,B 0,C 180,E1 -13380.459,E2 -13380.459} C_VEL
LIN {X 0,Y 360.973,Z 542.39,A -85,B 0,C 180,E1 -13382.458,E2 -13382.458} C_VEL
LIN {X 0,Y 359.039,Z 557.552,A -85,B 0,C 180,E1 -13385.811,E2 -13385.811} C_VEL
LIN {X 0,Y 362.715,Z 576.902,A -85,B 0,C 180,E1 -13386.772,E2 -13386.772} C_VEL
LIN {X 0,Y 365.028,Z 595.259,A -85,B 0,C 180,E1 -13387.542,E2 -13387.542} C_VEL
LIN {X 0,Y 365.61,Z 603.506,A -85,B 0,C 180,E1 -13387.841,E2 -13387.841} C_VEL
LIN {X 0,Y 363.14,Z 670.253,A -85,B 0,C 180,E1 -13389.576,E2 -13389.576} C_VEL
LIN {X 0,Y 362.223,Z 683.98,A -85,B 0,C 180,E1 -13390.152,E2 -13390.152} C_VEL
LIN {X 0,Y 360.947,Z 697.492,A -85,B 0,C 180,E1 -13390.966,E2 -13390.966} C_VEL
LIN {X 0,Y 359.633,Z 709.548,A -85,B 0,C 180,E1 -13391.927,E2 -13391.927} C_VEL
LIN {X 0,Y 357.644,Z 727.969,A -85,B 0,C 180,E1 -13393.739,E2 -13393.739} C_VEL
LIN {X 0,Y 356.714,Z 738.638,A -85,B 0,C 180,E1 -13395.061,E2 -13395.061} C_VEL
LIN {X 0,Y 355.682,Z 748.375,A -85,B 0,C 180,E1 -13396.575,E2 -13396.575} C_VEL
LIN {X 0,Y 354.709,Z 757.197,A -85,B 0,C 180,E1 -13398.283,E2 -13398.283} C_VEL
LIN {X 0,Y 354.077,Z 764.228,A -85,B 0,C 180,E1 -13399.999,E2 -13399.999} C_VEL
LIN {X 0,Y 353.613,Z 770.633,A -85,B 0,C 180,E1 -13402.003,E2 -13402.003} C_VEL
LIN {X 0,Y 353.388,Z 775.262,A -85,B 0,C 180,E1 -13403.921,E2 -13403.921} C_VEL
LIN {X 0,Y 353.306,Z 777.939,A -85,B 0,C 180,E1 -13405.436,E2 -13405.436} C_VEL
LIN {X 0,Y 353.264,Z 779.48,A -85,B 0,C 180,E1 -13406.578,E2 -13406.578} C_VEL
LIN {X 0,Y 353.236,Z 780.561,A -85,B 0,C 180,E1 -13407.72,E2 -13407.72} C_VEL
LIN {X 0,Y 353.252,Z 781.236,A -85,B 0,C 180,E1 -13408.86,E2 -13408.86} C_VEL
LIN {X 0,Y 353.27,Z 781.521,A -85,B 0,C 180,E1 -13410,E2 -13410} C_VEL
LIN {X 0,Y 353.236,Z 781.406,A -85,B 0,C 180,E1 -13411.14,E2 -13411.14} C_VEL
LIN {X 0,Y 353.235,Z 780.849,A -85,B 0,C 180,E1 -13412.28,E2 -13412.28} C_VEL
LIN {X 0,Y 353.265,Z 779.898,A -85,B 0,C 180,E1 -13413.422,E2 -13413.422} C_VEL
LIN {X 0,Y 353.308,Z 778.55,A -85,B 0,C 180,E1 -13414.564,E2 -13414.564} C_VEL
LIN {X 0,Y 353.388,Z 776.062,A -85,B 0,C 180,E1 -13416.079,E2 -13416.079} C_VEL
LIN {X 0,Y 353.634,Z 771.788,A -85,B 0,C 180,E1 -13417.996,E2 -13417.996} C_VEL
LIN {X 0,Y 354.032,Z 766.736,A -85,B 0,C 180,E1 -13419.714,E2 -13419.714} C_VEL
LIN {X 0,Y 354.643,Z 760.349,A -85,B 0,C 180,E1 -13421.43,E2 -13421.43} C_VEL
LIN {X 0,Y 355.625,Z 752.37,A -85,B 0,C 180,E1 -13423.136,E2 -13423.136} C_VEL
LIN {X 0,Y 356.535,Z 744.221,A -85,B 0,C 180,E1 -13424.556,E2 -13424.556} C_VEL
LIN {X 0,Y 357.66,Z 734.251,A -85,B 0,C 180,E1 -13425.968,E2 -13425.968} C_VEL
LIN {X 0,Y 358.731,Z 724.349,A -85,B 0,C 180,E1 -13427.089,E2 -13427.089} C_VEL
LIN {X 0,Y 359.969,Z 711.825,A -85,B 0,C 180,E1 -13428.202,E2 -13428.202} C_VEL
LIN {X 0,Y 360.878,Z 700.552,A -85,B 0,C 180,E1 -13428.964,E2 -13428.964} C_VEL
LIN {X 0,Y 361.732,Z 687.694,A -85,B 0,C 180,E1 -13429.581,E2 -13429.581} C_VEL
LIN {X 0,Y 362.238,Z 675.496,A -85,B 0,C 180,E1 -13429.958,E2 -13429.958} C_VEL
LIN {X 0,Y 363.435,Z 601.472,A -85,B 0,C 180,E1 -13431.432,E2 -13431.432} C_VEL
LIN {X 0,Y 359.012,Z 568.377,A -85,B 0,C 180,E1 -13432.422,E2 -13432.422} C_VEL
LIN {X 0,Y 357.784,Z 560.181,A -85,B 0,C 180,E1 -13432.7,E2 -13432.7} C_VEL
LIN {X 0,Y 357.547,Z 557.148,A -85,B 0,C 180,E1 -13432.932,E2 -13432.932} C_VEL
LIN {X 0,Y 359.317,Z 538.738,A -85,B 0,C 180,E1 -13436.734,E2 -13436.734} C_VEL
LIN {X 0,Y 358.868,Z 534.254,A -85,B 0,C 180,E1 -13437.717,E2 -13437.717} C_VEL
LIN {X 0,Y 355.918,Z 520.442,A -85,B 0,C 180,E1 -13440.89,E2 -13440.89} C_VEL
LIN {X 0,Y 354.846,Z 515.285,A -85,B 0,C 180,E1 -13442.135,E2 -13442.135} C_VEL
LIN {X 0,Y 354.819,Z 515.284,A -85,B 0,C 180,E1 -13445.699,E2 -13445.699} C_VEL
LIN {X 0,Y 354.821,Z 515.265,A -85,B 0,C 180,E1 -13449.423,E2 -13449.423} C_VEL
LIN {X 0,Y 354.785,Z 515.29,A -85,B 0,C 180,E1 -13452.867,E2 -13452.867} C_VEL
LIN {X 0,Y 354.798,Z 515.29,A -85,B 0,C 180,E1 -13456.108,E2 -13456.108} C_VEL
LIN {X 0,Y 354.819,Z 515.281,A -85,B 0,C 180,E1 -13459.183,E2 -13459.183} C_VEL
LIN {X 0,Y 354.808,Z 515.284,A -85,B 0,C 180,E1 -13462.401,E2 -13462.401} C_VEL
LIN {X 0,Y 354.806,Z 515.283,A -85,B 0,C 180,E1 -13464.94,E2 -13464.94} C_VEL
LIN {X 0,Y 354.787,Z 515.282,A -85,B 0,C 180,E1 -13468.405,E2 -13468.405} C_VEL
LIN {X 0,Y 354.847,Z 515.283,A -85,B 0,C 180,E1 -13471.619,E2 -13471.619} C_VEL
LIN {X 0,Y 354.892,Z 515.271,A -85,B 0,C 180,E1 -13474.172,E2 -13474.172} C_VEL
LIN {X 0,Y 354.808,Z 515.282,A -85,B 0,C 180,E1 -13477.892,E2 -13477.892} C_VEL
LIN {X 0,Y 354.915,Z 515.263,A -85,B 0,C 180,E1 -13481.891,E2 -13481.891} C_VEL
LIN {X 0,Y 354.935,Z 515.268,A -85,B 0,C 180,E1 -13485.981,E2 -13485.981} C_VEL
LIN {X 0,Y 354.975,Z 515.257,A -85,B 0,C 180,E1 -13489.736,E2 -13489.736} C_VEL
LIN {X 0,Y 355.124,Z 515.234,A -85,B 0,C 180,E1 -13493.181,E2 -13493.181} C_VEL
LIN {X 0,Y 355.238,Z 515.226,A -85,B 0,C 180,E1 -13497.733,E2 -13497.733} C_VEL
LIN {X 0,Y 355.391,Z 515.188,A -85,B 0,C 180,E1 -13500,E2 -13500} C_VEL
LIN {X 0,Y 355.239,Z 515.226,A -85,B 0,C 180,E1 -13502.268,E2 -13502.268} C_VEL
LIN {X 0,Y 355.122,Z 515.237,A -85,B 0,C 180,E1 -13506.82,E2 -13506.82} C_VEL
LIN {X 0,Y 354.971,Z 515.258,A -85,B 0,C 180,E1 -13510.265,E2 -13510.265} C_VEL
LIN {X 0,Y 354.935,Z 515.266,A -85,B 0,C 180,E1 -13514.019,E2 -13514.019} C_VEL
LIN {X 0,Y 354.916,Z 515.268,A -85,B 0,C 180,E1 -13518.109,E2 -13518.109} C_VEL
LIN {X 0,Y 354.828,Z 515.277,A -85,B 0,C 180,E1 -13522.107,E2 -13522.107} C_VEL
LIN {X 0,Y 354.894,Z 515.276,A -85,B 0,C 180,E1 -13525.828,E2 -13525.828} C_VEL
LIN {X 0,Y 354.85,Z 515.27,A -85,B 0,C 180,E1 -13529.679,E2 -13529.679} C_VEL
LIN {X 0,Y 354.827,Z 515.281,A -85,B 0,C 180,E1 -13533.683,E2 -13533.683} C_VEL
LIN {X 0,Y 354.795,Z 515.289,A -85,B 0,C 180,E1 -13536.46,E2 -13536.46} C_VEL
LIN {X 0,Y 354.821,Z 515.282,A -85,B 0,C 180,E1 -13539.425,E2 -13539.425} C_VEL
LIN {X 0,Y 354.786,Z 515.291,A -85,B 0,C 180,E1 -13542.868,E2 -13542.868} C_VEL
LIN {X 0,Y 354.775,Z 515.293,A -85,B 0,C 180,E1 -13546.106,E2 -13546.106} C_VEL
LIN {X 0,Y 354.787,Z 515.289,A -85,B 0,C 180,E1 -13549.18,E2 -13549.18} C_VEL
LIN {X 0,Y 354.807,Z 515.286,A -85,B 0,C 180,E1 -13552.404,E2 -13552.404} C_VEL
LIN {X 0,Y 354.812,Z 515.278,A -85,B 0,C 180,E1 -13554.942,E2 -13554.942} C_VEL
LIN {X 0,Y 354.85,Z 515.307,A -85,B 0,C 180,E1 -13558.185,E2 -13558.185} C_VEL
LIN {X 0,Y 358.111,Z 528.816,A -85,B 0,C 180,E1 -13561.263,E2 -13561.263} C_VEL
LIN {X 0,Y 359.676,Z 536.724,A -85,B 0,C 180,E1 -13562.981,E2 -13562.981} C_VEL
LIN {X 0,Y 359.559,Z 543.154,A -85,B 0,C 180,E1 -13564.241,E2 -13564.241} C_VEL
LIN {X 0,Y 359.205,Z 549.088,A -85,B 0,C 180,E1 -13565.347,E2 -13565.347} C_VEL
LIN {X 0,Y 364.375,Z 575.74,A -85,B 0,C 180,E1 -13566.273,E2 -13566.273} C_VEL
LIN {X 0,Y 362.818,Z 659.436,A -85,B 0,C 180,E1 -13567.957,E2 -13567.957} C_VEL
LIN {X 0,Y 362.237,Z 672.631,A -85,B 0,C 180,E1 -13568.437,E2 -13568.437} C_VEL
LIN {X 0,Y 361.543,Z 685.25,A -85,B 0,C 180,E1 -13569.143,E2 -13569.143} C_VEL
LIN {X 0,Y 360.558,Z 697.409,A -85,B 0,C 180,E1 -13570.056,E2 -13570.056} C_VEL
LIN {X 0,Y 359.383,Z 708.832,A -85,B 0,C 180,E1 -13571.176,E2 -13571.176} C_VEL
LIN {X 0,Y 358.139,Z 719.095,A -85,B 0,C 180,E1 -13572.44,E2 -13572.44} C_VEL
LIN {X 0,Y 357.131,Z 727.503,A -85,B 0,C 180,E1 -13573.715,E2 -13573.715} C_VEL
LIN {X 0,Y 356.161,Z 735.655,A -85,B 0,C 180,E1 -13575.22,E2 -13575.22} C_VEL
LIN {X 0,Y 355.271,Z 743.898,A -85,B 0,C 180,E1 -13577.142,E2 -13577.142} C_VEL
LIN {X 0,Y 354.359,Z 750.603,A -85,B 0,C 180,E1 -13579.14,E2 -13579.14} C_VEL
LIN {X 0,Y 353.889,Z 754.991,A -85,B 0,C 180,E1 -13580.859,E2 -13580.859} C_VEL
LIN {X 0,Y 353.659,Z 757.294,A -85,B 0,C 180,E1 -13582.004,E2 -13582.004} C_VEL
LIN {X 0,Y 353.437,Z 760.1,A -85,B 0,C 180,E1 -13583.851,E2 -13583.851} C_VEL
LIN {X 0,Y 353.311,Z 761.644,A -85,B 0,C 180,E1 -13585.436,E2 -13585.436} C_VEL
LIN {X 0,Y 353.213,Z 762.524,A -85,B 0,C 180,E1 -13587.719,E2 -13587.719} C_VEL
LIN {X 0,Y 353.23,Z 762.361,A -85,B 0,C 180,E1 -13588.86,E2 -13588.86} C_VEL
LIN {X 0,Y 353.265,Z 761.789,A -85,B 0,C 180,E1 -13590,E2 -13590} C_VEL
LIN {X 0,Y 353.427,Z 759.495,A -85,B 0,C 180,E1 -13592.279,E2 -13592.279} C_VEL
LIN {X 0,Y 353.648,Z 756.654,A -85,B 0,C 180,E1 -13593.988,E2 -13593.988} C_VEL
LIN {X 0,Y 353.977,Z 752.793,A -85,B 0,C 180,E1 -13595.697,E2 -13595.697} C_VEL
LIN {X 0,Y 354.536,Z 747.051,A -85,B 0,C 180,E1 -13597.622,E2 -13597.622} C_VEL
LIN {X 0,Y 355.227,Z 740.294,A -85,B 0,C 180,E1 -13599.394,E2 -13599.394} C_VEL
LIN {X 0,Y 356.158,Z 732.181,A -85,B 0,C 180,E1 -13601.092,E2 -13601.092} C_VEL
LIN {X 0,Y 357.118,Z 723.82,A -85,B 0,C 180,E1 -13602.502,E2 -13602.502} C_VEL
LIN {X 0,Y 358.16,Z 713.561,A -85,B 0,C 180,E1 -13603.908,E2 -13603.908} C_VEL
LIN {X 0,Y 359.182,Z 703.422,A -85,B 0,C 180,E1 -13605.026,E2 -13605.026} C_VEL
LIN {X 0,Y 360.102,Z 692.279,A -85,B 0,C 180,E1 -13606.002,E2 -13606.002} C_VEL
LIN {X 0,Y 361.047,Z 679.687,A -85,B 0,C 180,E1 -13606.831,E2 -13606.831} C_VEL
LIN {X 0,Y 361.562,Z 667.081,A -85,B 0,C 180,E1 -13607.435,E2 -13607.435} C_VEL
LIN {X 0,Y 361.957,Z 654.088,A -85,B 0,C 180,E1 -13607.818,E2 -13607.818} C_VEL
LIN {X 0,Y 362.338,Z 637.26,A -85,B 0,C 180,E1 -13608.146,E2 -13608.146} C_VEL
LIN {X 0,Y 361.811,Z 631.45,A -85,B 0,C 180,E1 -13608.296,E2 -13608.296} C_VEL
LIN {X 0,Y 356.672,Z 612.768,A -85,B 0,C 180,E1 -13608.982,E2 -13608.982} C_VEL
LIN {X 0,Y 356.187,Z 606.958,A -85,B 0,C 180,E1 -13609.133,E2 -13609.133} C_VEL
LIN {X 0,Y 356.618,Z 576.331,A -85,B 0,C 180,E1 -13609.755,E2 -13609.755} C_VEL
LIN {X 0,Y 352.02,Z 550.529,A -85,B 0,C 180,E1 -13610.598,E2 -13610.598} C_VEL
LIN {X 0,Y 351.803,Z 549.002,A -85,B 0,C 180,E1 -13610.69,E2 -13610.69} C_VEL
LIN {X 0,Y 352.211,Z 536.636,A -85,B 0,C 180,E1 -13613.059,E2 -13613.059} C_VEL
LIN {X 0,Y 349.806,Z 524.586,A -85,B 0,C 180,E1 -13615.707,E2 -13615.707} C_VEL
LIN {X 0,Y 347.868,Z 516.153,A -85,B 0,C 180,E1 -13617.619,E2 -13617.619} C_VEL
LIN {X 0,Y 347.765,Z 516.17,A -85,B 0,C 180,E1 -13620.346,E2 -13620.346} C_VEL
LIN {X 0,Y 347.745,Z 516.167,A -85,B 0,C 180,E1 -13624.463,E2 -13624.463} C_VEL
LIN {X 0,Y 347.774,Z 516.164,A -85,B 0,C 180,E1 -13627.988,E2 -13627.988} C_VEL
LIN {X 0,Y 347.782,Z 516.163,A -85,B 0,C 180,E1 -13631.608,E2 -13631.608} C_VEL
LIN {X 0,Y 347.794,Z 516.15,A -85,B 0,C 180,E1 -13635.011,E2 -13635.011} C_VEL
LIN {X 0,Y 347.748,Z 516.169,A -85,B 0,C 180,E1 -13638.396,E2 -13638.396} C_VEL
LIN {X 0,Y 347.776,Z 516.184,A -85,B 0,C 180,E1 -13642.159,E2 -13642.159} C_VEL
LIN {X 0,Y 355.253,Z 537.083,A -85,B 0,C 180,E1 -13643.083,E2 -13643.083} C_VEL
LIN {X 0,Y 353.258,Z 619.174,A -85,B 0,C 180,E1 -13645.133,E2 -13645.133} C_VEL
LIN {X 0,Y 352.848,Z 631.958,A -85,B 0,C 180,E1 -13645.672,E2 -13645.672} C_VEL
LIN {X 0,Y 352.333,Z 643.347,A -85,B 0,C 180,E1 -13646.343,E2 -13646.343} C_VEL
LIN {X 0,Y 351.515,Z 655.99,A -85,B 0,C 180,E1 -13647.328,E2 -13647.328} C_VEL
LIN {X 0,Y 350.609,Z 668.482,A -85,B 0,C 180,E1 -13648.589,E2 -13648.589} C_VEL
LIN {X 0,Y 349.75,Z 679.502,A -85,B 0,C 180,E1 -13650.01,E2 -13650.01} C_VEL
LIN {X 0,Y 348.958,Z 688.437,A -85,B 0,C 180,E1 -13651.423,E2 -13651.423} C_VEL
LIN {X 0,Y 348.279,Z 696.616,A -85,B 0,C 180,E1 -13653.001,E2 -13653.001} C_VEL
LIN {X 0,Y 347.636,Z 704.377,A -85,B 0,C 180,E1 -13654.878,E2 -13654.878} C_VEL
